        ToWin32ErrorCode := Win32ErrorCodes.ERROR_DS_DRA_OUT_OF_MEM;
    8447:
        ToWin32ErrorCode := Win32ErrorCodes.ERROR_DS_DRA_MAIL_PROBLEM;
    8448:
        ToWin32ErrorCode := Win32ErrorCodes.ERROR_DS_DRA_REF_ALREADY_EXISTS;
    8449:
        ToWin32ErrorCode := Win32ErrorCodes.ERROR_DS_DRA_REF_NOT_FOUND;
    8450:
        ToWin32ErrorCode := Win32ErrorCodes.ERROR_DS_DRA_OBJ_IS_REP_SOURCE;
    8451:
        ToWin32ErrorCode := Win32ErrorCodes.ERROR_DS_DRA_DB_ERROR;
    8452:
        ToWin32ErrorCode := Win32ErrorCodes.ERROR_DS_DRA_NO_REPLICA;
    8453:
        ToWin32ErrorCode := Win32ErrorCodes.ERROR_DS_DRA_ACCESS_DENIED;
    8454:
        ToWin32ErrorCode := Win32ErrorCodes.ERROR_DS_DRA_NOT_SUPPORTED;
    8455:
        ToWin32ErrorCode := Win32ErrorCodes.ERROR_DS_DRA_RPC_CANCELLED;
    8456:
        ToWin32ErrorCode := Win32ErrorCodes.ERROR_DS_DRA_SOURCE_DISABLED;
    8457:
        ToWin32ErrorCode := Win32ErrorCodes.ERROR_DS_DRA_SINK_DISABLED;
    8458:
        ToWin32ErrorCode := Win32ErrorCodes.ERROR_DS_DRA_NAME_COLLISION;
    8459:
        ToWin32ErrorCode := Win32ErrorCodes.ERROR_DS_DRA_SOURCE_REINSTALLED;
    8460:
        ToWin32ErrorCode := Win32ErrorCodes.ERROR_DS_DRA_MISSING_PARENT;
    8461:
        ToWin32ErrorCode := Win32ErrorCodes.ERROR_DS_DRA_PREEMPTED;
    8462:
        ToWin32ErrorCode := Win32ErrorCodes.ERROR_DS_DRA_ABANDON_SYNC;
    8463:
        ToWin32ErrorCode := Win32ErrorCodes.ERROR_DS_DRA_SHUTDOWN;
    8464:
        ToWin32ErrorCode := Win32ErrorCodes.ERROR_DS_DRA_INCOMPATIBLE_PARTIAL_SET;
    8465:
        ToWin32ErrorCode := Win32ErrorCodes.ERROR_DS_DRA_SOURCE_IS_PARTIAL_REPLICA;
    8466:
        ToWin32ErrorCode := Win32ErrorCodes.ERROR_DS_DRA_EXTN_CONNECTION_FAILED;
    8467:
        ToWin32ErrorCode := Win32ErrorCodes.ERROR_DS_INSTALL_SCHEMA_MISMATCH;
    8468:
        ToWin32ErrorCode := Win32ErrorCodes.ERROR_DS_DUP_LINK_ID;
    8469:
        ToWin32ErrorCode := Win32ErrorCodes.ERROR_DS_NAME_ERROR_RESOLVING;
    8470:
        ToWin32ErrorCode := Win32ErrorCodes.ERROR_DS_NAME_ERROR_NOT_FOUND;
    8471:
        ToWin32ErrorCode := Win32ErrorCodes.ERROR_DS_NAME_ERROR_NOT_UNIQUE;
    8472:
        ToWin32ErrorCode := Win32ErrorCodes.ERROR_DS_NAME_ERROR_NO_MAPPING;
    8473:
        ToWin32ErrorCode := Win32ErrorCodes.ERROR_DS_NAME_ERROR_DOMAIN_ONLY;
    8474:
        ToWin32ErrorCode := Win32ErrorCodes.ERROR_DS_NAME_ERROR_NO_SYNTACTICAL_MAPPING;
    8475:
        ToWin32ErrorCode := Win32ErrorCodes.ERROR_DS_CONSTRUCTED_ATT_MOD;
    8476:
        ToWin32ErrorCode := Win32ErrorCodes.ERROR_DS_WRONG_OM_OBJ_CLASS;
    8477:
        ToWin32ErrorCode := Win32ErrorCodes.ERROR_DS_DRA_REPL_PENDING;
    8478:
        ToWin32ErrorCode := Win32ErrorCodes.ERROR_DS_DS_REQUIRED;
    8479:
        ToWin32ErrorCode := Win32ErrorCodes.ERROR_DS_INVALID_LDAP_DISPLAY_NAME;
    8480:
        ToWin32ErrorCode := Win32ErrorCodes.ERROR_DS_NON_BASE_SEARCH;
    8481:
        ToWin32ErrorCode := Win32ErrorCodes.ERROR_DS_CANT_RETRIEVE_ATTS;
    8482:
        ToWin32ErrorCode := Win32ErrorCodes.ERROR_DS_BACKLINK_WITHOUT_LINK;
    8483:
        ToWin32ErrorCode := Win32ErrorCodes.ERROR_DS_EPOCH_MISMATCH;
    8484:
        ToWin32ErrorCode := Win32ErrorCodes.ERROR_DS_SRC_NAME_MISMATCH;
    8485:
        ToWin32ErrorCode := Win32ErrorCodes.ERROR_DS_SRC_AND_DST_NC_IDENTICAL;
    8486:
        ToWin32ErrorCode := Win32ErrorCodes.ERROR_DS_DST_NC_MISMATCH;
    8487:
        ToWin32ErrorCode := Win32ErrorCodes.ERROR_DS_NOT_AUTHORITIVE_FOR_DST_NC;
    8488:
        ToWin32ErrorCode := Win32ErrorCodes.ERROR_DS_SRC_GUID_MISMATCH;
    8489:
        ToWin32ErrorCode := Win32ErrorCodes.ERROR_DS_CANT_MOVE_DELETED_OBJECT;
    8490:
        ToWin32ErrorCode := Win32ErrorCodes.ERROR_DS_PDC_OPERATION_IN_PROGRESS;
    8491:
        ToWin32ErrorCode := Win32ErrorCodes.ERROR_DS_CROSS_DOMAIN_CLEANUP_REQD;
    8492:
        ToWin32ErrorCode := Win32ErrorCodes.ERROR_DS_ILLEGAL_XDOM_MOVE_OPERATION;
    8493:
        ToWin32ErrorCode := Win32ErrorCodes.ERROR_DS_CANT_WITH_ACCT_GROUP_MEMBERSHPS;
    8494:
        ToWin32ErrorCode := Win32ErrorCodes.ERROR_DS_NC_MUST_HAVE_NC_PARENT;
    8495:
        ToWin32ErrorCode := Win32ErrorCodes.ERROR_DS_CR_IMPOSSIBLE_TO_VALIDATE;
    8496:
        ToWin32ErrorCode := Win32ErrorCodes.ERROR_DS_DST_DOMAIN_NOT_NATIVE;
    8497:
        ToWin32ErrorCode := Win32ErrorCodes.ERROR_DS_MISSING_INFRASTRUCTURE_CONTAINER;
    8498:
        ToWin32ErrorCode := Win32ErrorCodes.ERROR_DS_CANT_MOVE_ACCOUNT_GROUP;
    8499:
        ToWin32ErrorCode := Win32ErrorCodes.ERROR_DS_CANT_MOVE_RESOURCE_GROUP;
    8500:
        ToWin32ErrorCode := Win32ErrorCodes.ERROR_DS_INVALID_SEARCH_FLAG;
    8501:
        ToWin32ErrorCode := Win32ErrorCodes.ERROR_DS_NO_TREE_DELETE_ABOVE_NC;
    8502:
        ToWin32ErrorCode := Win32ErrorCodes.ERROR_DS_COULDNT_LOCK_TREE_FOR_DELETE;
    8503:
        ToWin32ErrorCode := Win32ErrorCodes.ERROR_DS_COULDNT_IDENTIFY_OBJECTS_FOR_TREE_DELETE;
    8504:
        ToWin32ErrorCode := Win32ErrorCodes.ERROR_DS_SAM_INIT_FAILURE;
    8505:
        ToWin32ErrorCode := Win32ErrorCodes.ERROR_DS_SENSITIVE_GROUP_VIOLATION;
    8506:
        ToWin32ErrorCode := Win32ErrorCodes.ERROR_DS_CANT_MOD_PRIMARYGROUPID;
    8507:
        ToWin32ErrorCode := Win32ErrorCodes.ERROR_DS_ILLEGAL_BASE_SCHEMA_MOD;
    8508:
        ToWin32ErrorCode := Win32ErrorCodes.ERROR_DS_NONSAFE_SCHEMA_CHANGE;
    8509:
        ToWin32ErrorCode := Win32ErrorCodes.ERROR_DS_SCHEMA_UPDATE_DISALLOWED;
    8510:
        ToWin32ErrorCode := Win32ErrorCodes.ERROR_DS_CANT_CREATE_UNDER_SCHEMA;
    8511:
        ToWin32ErrorCode := Win32ErrorCodes.ERROR_DS_INSTALL_NO_SRC_SCH_VERSION;
    8512:
        ToWin32ErrorCode := Win32ErrorCodes.ERROR_DS_INSTALL_NO_SCH_VERSION_IN_INIFILE;
    8513:
        ToWin32ErrorCode := Win32ErrorCodes.ERROR_DS_INVALID_GROUP_TYPE;
    8514:
        ToWin32ErrorCode := Win32ErrorCodes.ERROR_DS_NO_NEST_GLOBALGROUP_IN_MIXEDDOMAIN;
    8515:
        ToWin32ErrorCode := Win32ErrorCodes.ERROR_DS_NO_NEST_LOCALGROUP_IN_MIXEDDOMAIN;
    8516:
        ToWin32ErrorCode := Win32ErrorCodes.ERROR_DS_GLOBAL_CANT_HAVE_LOCAL_MEMBER;
    8517:
        ToWin32ErrorCode := Win32ErrorCodes.ERROR_DS_GLOBAL_CANT_HAVE_UNIVERSAL_MEMBER;
    8518:
        ToWin32ErrorCode := Win32ErrorCodes.ERROR_DS_UNIVERSAL_CANT_HAVE_LOCAL_MEMBER;
    8519:
        ToWin32ErrorCode := Win32ErrorCodes.ERROR_DS_GLOBAL_CANT_HAVE_CROSSDOMAIN_MEMBER;
    8520:
        ToWin32ErrorCode := Win32ErrorCodes.ERROR_DS_LOCAL_CANT_HAVE_CROSSDOMAIN_LOCAL_MEMBER;
    8521:
        ToWin32ErrorCode := Win32ErrorCodes.ERROR_DS_HAVE_PRIMARY_MEMBERS;
    8522:
        ToWin32ErrorCode := Win32ErrorCodes.ERROR_DS_STRING_SD_CONVERSION_FAILED;
    8523:
        ToWin32ErrorCode := Win32ErrorCodes.ERROR_DS_NAMING_MASTER_GC;
    8524:
        ToWin32ErrorCode := Win32ErrorCodes.ERROR_DS_LOOKUP_FAILURE;
    8525:
        ToWin32ErrorCode := Win32ErrorCodes.ERROR_DS_COULDNT_UPDATE_SPNS;
    8526:
        ToWin32ErrorCode := Win32ErrorCodes.ERROR_DS_CANT_RETRIEVE_SD;
    8527:
        ToWin32ErrorCode := Win32ErrorCodes.ERROR_DS_KEY_NOT_UNIQUE;
    8528:
        ToWin32ErrorCode := Win32ErrorCodes.ERROR_DS_WRONG_LINKED_ATT_SYNTAX;
    8529:
        ToWin32ErrorCode := Win32ErrorCodes.ERROR_DS_SAM_NEED_BOOTKEY_PASSWORD;
    8530:
        ToWin32ErrorCode := Win32ErrorCodes.ERROR_DS_SAM_NEED_BOOTKEY_FLOPPY;
    8531:
        ToWin32ErrorCode := Win32ErrorCodes.ERROR_DS_CANT_START;
    8532:
        ToWin32ErrorCode := Win32ErrorCodes.ERROR_DS_INIT_FAILURE;
    8533:
        ToWin32ErrorCode := Win32ErrorCodes.ERROR_DS_NO_PKT_PRIVACY_ON_CONNECTION;
    8534:
        ToWin32ErrorCode := Win32ErrorCodes.ERROR_DS_SOURCE_DOMAIN_IN_FOREST;
    8535:
        ToWin32ErrorCode := Win32ErrorCodes.ERROR_DS_DESTINATION_DOMAIN_NOT_IN_FOREST;
    8536:
        ToWin32ErrorCode := Win32ErrorCodes.ERROR_DS_DESTINATION_AUDITING_NOT_ENABLED;
    8537:
        ToWin32ErrorCode := Win32ErrorCodes.ERROR_DS_CANT_FIND_DC_FOR_SRC_DOMAIN;
    8538:
        ToWin32ErrorCode := Win32ErrorCodes.ERROR_DS_SRC_OBJ_NOT_GROUP_OR_USER;
    8539:
        ToWin32ErrorCode := Win32ErrorCodes.ERROR_DS_SRC_SID_EXISTS_IN_FOREST;
    8540:
        ToWin32ErrorCode := Win32ErrorCodes.ERROR_DS_SRC_AND_DST_OBJECT_CLASS_MISMATCH;
    8541:
        ToWin32ErrorCode := Win32ErrorCodes.ERROR_SAM_INIT_FAILURE;
    8542:
        ToWin32ErrorCode := Win32ErrorCodes.ERROR_DS_DRA_SCHEMA_INFO_SHIP;
    8543:
        ToWin32ErrorCode := Win32ErrorCodes.ERROR_DS_DRA_SCHEMA_CONFLICT;
    8544:
        ToWin32ErrorCode := Win32ErrorCodes.ERROR_DS_DRA_EARLIER_SCHEMA_CONLICT;
    8545:
        ToWin32ErrorCode := Win32ErrorCodes.ERROR_DS_DRA_OBJ_NC_MISMATCH;
    8546:
        ToWin32ErrorCode := Win32ErrorCodes.ERROR_DS_NC_STILL_HAS_DSAS;
    8547:
        ToWin32ErrorCode := Win32ErrorCodes.ERROR_DS_GC_REQUIRED;
    8548:
        ToWin32ErrorCode := Win32ErrorCodes.ERROR_DS_LOCAL_MEMBER_OF_LOCAL_ONLY;
    8549:
        ToWin32ErrorCode := Win32ErrorCodes.ERROR_DS_NO_FPO_IN_UNIVERSAL_GROUPS;
    8550:
        ToWin32ErrorCode := Win32ErrorCodes.ERROR_DS_CANT_ADD_TO_GC;
    8551:
        ToWin32ErrorCode := Win32ErrorCodes.ERROR_DS_NO_CHECKPOINT_WITH_PDC;
    8552:
        ToWin32ErrorCode := Win32ErrorCodes.ERROR_DS_SOURCE_AUDITING_NOT_ENABLED;
    8553:
        ToWin32ErrorCode := Win32ErrorCodes.ERROR_DS_CANT_CREATE_IN_NONDOMAIN_NC;
    8554:
        ToWin32ErrorCode := Win32ErrorCodes.ERROR_DS_INVALID_NAME_FOR_SPN;
    8555:
        ToWin32ErrorCode := Win32ErrorCodes.ERROR_DS_FILTER_USES_CONTRUCTED_ATTRS;
    8556:
        ToWin32ErrorCode := Win32ErrorCodes.ERROR_DS_UNICODEPWD_NOT_IN_QUOTES;
    8557:
        ToWin32ErrorCode := Win32ErrorCodes.ERROR_DS_MACHINE_ACCOUNT_QUOTA_EXCEEDED;
    8558:
        ToWin32ErrorCode := Win32ErrorCodes.ERROR_DS_MUST_BE_RUN_ON_DST_DC;
    8559:
        ToWin32ErrorCode := Win32ErrorCodes.ERROR_DS_SRC_DC_MUST_BE_SP4_OR_GREATER;
    8560:
        ToWin32ErrorCode := Win32ErrorCodes.ERROR_DS_CANT_TREE_DELETE_CRITICAL_OBJ;
    8561:
        ToWin32ErrorCode := Win32ErrorCodes.ERROR_DS_INIT_FAILURE_CONSOLE;
    8562:
        ToWin32ErrorCode := Win32ErrorCodes.ERROR_DS_SAM_INIT_FAILURE_CONSOLE;
    8563:
        ToWin32ErrorCode := Win32ErrorCodes.ERROR_DS_FOREST_VERSION_TOO_HIGH;
    8564:
        ToWin32ErrorCode := Win32ErrorCodes.ERROR_DS_DOMAIN_VERSION_TOO_HIGH;
    8565:
        ToWin32ErrorCode := Win32ErrorCodes.ERROR_DS_FOREST_VERSION_TOO_LOW;
    8566:
        ToWin32ErrorCode := Win32ErrorCodes.ERROR_DS_DOMAIN_VERSION_TOO_LOW;
    8567:
        ToWin32ErrorCode := Win32ErrorCodes.ERROR_DS_INCOMPATIBLE_VERSION;
    8568:
        ToWin32ErrorCode := Win32ErrorCodes.ERROR_DS_LOW_DSA_VERSION;
    8569:
        ToWin32ErrorCode := Win32ErrorCodes.ERROR_DS_NO_BEHAVIOR_VERSION_IN_MIXEDDOMAIN;
    8570:
        ToWin32ErrorCode := Win32ErrorCodes.ERROR_DS_NOT_SUPPORTED_SORT_ORDER;
    8571:
        ToWin32ErrorCode := Win32ErrorCodes.ERROR_DS_NAME_NOT_UNIQUE;
    8572:
        ToWin32ErrorCode := Win32ErrorCodes.ERROR_DS_MACHINE_ACCOUNT_CREATED_PRENT4;
    8573:
        ToWin32ErrorCode := Win32ErrorCodes.ERROR_DS_OUT_OF_VERSION_STORE;
    8574:
        ToWin32ErrorCode := Win32ErrorCodes.ERROR_DS_INCOMPATIBLE_CONTROLS_USED;
    8575:
        ToWin32ErrorCode := Win32ErrorCodes.ERROR_DS_NO_REF_DOMAIN;
    8576:
        ToWin32ErrorCode := Win32ErrorCodes.ERROR_DS_RESERVED_LINK_ID;
    8577:
        ToWin32ErrorCode := Win32ErrorCodes.ERROR_DS_LINK_ID_NOT_AVAILABLE;
    8578:
        ToWin32ErrorCode := Win32ErrorCodes.ERROR_DS_AG_CANT_HAVE_UNIVERSAL_MEMBER;
    8579:
        ToWin32ErrorCode := Win32ErrorCodes.ERROR_DS_MODIFYDN_DISALLOWED_BY_INSTANCE_TYPE;
    8580:
        ToWin32ErrorCode := Win32ErrorCodes.ERROR_DS_NO_OBJECT_MOVE_IN_SCHEMA_NC;
    8581:
        ToWin32ErrorCode := Win32ErrorCodes.ERROR_DS_MODIFYDN_DISALLOWED_BY_FLAG;
    8582:
        ToWin32ErrorCode := Win32ErrorCodes.ERROR_DS_MODIFYDN_WRONG_GRANDPARENT;
    8583:
        ToWin32ErrorCode := Win32ErrorCodes.ERROR_DS_NAME_ERROR_TRUST_REFERRAL;
    8584:
        ToWin32ErrorCode := Win32ErrorCodes.ERROR_NOT_SUPPORTED_ON_STANDARD_SERVER;
    8585:
        ToWin32ErrorCode := Win32ErrorCodes.ERROR_DS_CANT_ACCESS_REMOTE_PART_OF_AD;
    8586:
        ToWin32ErrorCode := Win32ErrorCodes.ERROR_DS_CR_IMPOSSIBLE_TO_VALIDATE_V2;
    8587:
        ToWin32ErrorCode := Win32ErrorCodes.ERROR_DS_THREAD_LIMIT_EXCEEDED;
    8588:
        ToWin32ErrorCode := Win32ErrorCodes.ERROR_DS_NOT_CLOSEST;
    9001:
        ToWin32ErrorCode := Win32ErrorCodes.DNS_ERROR_RCODE_FORMAT_ERROR;
    9002:
        ToWin32ErrorCode := Win32ErrorCodes.DNS_ERROR_RCODE_SERVER_FAILURE;
    9003:
        ToWin32ErrorCode := Win32ErrorCodes.DNS_ERROR_RCODE_NAME_ERROR;
    9004:
        ToWin32ErrorCode := Win32ErrorCodes.DNS_ERROR_RCODE_NOT_IMPLEMENTED;
    9005:
        ToWin32ErrorCode := Win32ErrorCodes.DNS_ERROR_RCODE_REFUSED;
    9006:
        ToWin32ErrorCode := Win32ErrorCodes.DNS_ERROR_RCODE_YXDOMAIN;
    9007:
        ToWin32ErrorCode := Win32ErrorCodes.DNS_ERROR_RCODE_YXRRSET;
    9008:
        ToWin32ErrorCode := Win32ErrorCodes.DNS_ERROR_RCODE_NXRRSET;
    9009:
        ToWin32ErrorCode := Win32ErrorCodes.DNS_ERROR_RCODE_NOTAUTH;
    9010:
        ToWin32ErrorCode := Win32ErrorCodes.DNS_ERROR_RCODE_NOTZONE;
    9016:
        ToWin32ErrorCode := Win32ErrorCodes.DNS_ERROR_RCODE_BADSIG;
    9017:
        ToWin32ErrorCode := Win32ErrorCodes.DNS_ERROR_RCODE_BADKEY;
    9018:
        ToWin32ErrorCode := Win32ErrorCodes.DNS_ERROR_RCODE_BADTIME;
    9501:
        ToWin32ErrorCode := Win32ErrorCodes.DNS_INFO_NO_RECORDS;
    9502:
        ToWin32ErrorCode := Win32ErrorCodes.DNS_ERROR_BAD_PACKET;
    9503:
        ToWin32ErrorCode := Win32ErrorCodes.DNS_ERROR_NO_PACKET;
    9504:
        ToWin32ErrorCode := Win32ErrorCodes.DNS_ERROR_RCODE;
    9505:
        ToWin32ErrorCode := Win32ErrorCodes.DNS_ERROR_UNSECURE_PACKET;
    9551:
        ToWin32ErrorCode := Win32ErrorCodes.DNS_ERROR_INVALID_TYPE;
    9552:
        ToWin32ErrorCode := Win32ErrorCodes.DNS_ERROR_INVALID_IP_ADDRESS;
    9553:
        ToWin32ErrorCode := Win32ErrorCodes.DNS_ERROR_INVALID_PROPERTY;
    9554:
        ToWin32ErrorCode := Win32ErrorCodes.DNS_ERROR_TRY_AGAIN_LATER;
    9555:
        ToWin32ErrorCode := Win32ErrorCodes.DNS_ERROR_NOT_UNIQUE;
    9556:
        ToWin32ErrorCode := Win32ErrorCodes.DNS_ERROR_NON_RFC_NAME;
    9557:
        ToWin32ErrorCode := Win32ErrorCodes.DNS_STATUS_FQDN;
    9558:
        ToWin32ErrorCode := Win32ErrorCodes.DNS_STATUS_DOTTED_NAME;
    9559:
        ToWin32ErrorCode := Win32ErrorCodes.DNS_STATUS_SINGLE_PART_NAME;
    9560:
        ToWin32ErrorCode := Win32ErrorCodes.DNS_ERROR_INVALID_NAME_CHAR;
    9561:
        ToWin32ErrorCode := Win32ErrorCodes.DNS_ERROR_NUMERIC_NAME;
    9601:
        ToWin32ErrorCode := Win32ErrorCodes.DNS_ERROR_ZONE_DOES_NOT_EXIST;
    9602:
        ToWin32ErrorCode := Win32ErrorCodes.DNS_ERROR_NO_ZONE_INFO;
    9603:
        ToWin32ErrorCode := Win32ErrorCodes.DNS_ERROR_INVALID_ZONE_OPERATION;
    9604:
        ToWin32ErrorCode := Win32ErrorCodes.DNS_ERROR_ZONE_CONFIGURATION_ERROR;
    9605:
        ToWin32ErrorCode := Win32ErrorCodes.DNS_ERROR_ZONE_HAS_NO_SOA_RECORD;
    9606:
        ToWin32ErrorCode := Win32ErrorCodes.DNS_ERROR_ZONE_HAS_NO_NS_RECORDS;
    9607:
        ToWin32ErrorCode := Win32ErrorCodes.DNS_ERROR_ZONE_LOCKED;
    9608:
        ToWin32ErrorCode := Win32ErrorCodes.DNS_ERROR_ZONE_CREATION_FAILED;
    9609:
        ToWin32ErrorCode := Win32ErrorCodes.DNS_ERROR_ZONE_ALREADY_EXISTS;
    9610:
        ToWin32ErrorCode := Win32ErrorCodes.DNS_ERROR_AUTOZONE_ALREADY_EXISTS;
    9611:
        ToWin32ErrorCode := Win32ErrorCodes.DNS_ERROR_INVALID_ZONE_TYPE;
    9612:
        ToWin32ErrorCode := Win32ErrorCodes.DNS_ERROR_SECONDARY_REQUIRES_MASTER_IP;
    9613:
        ToWin32ErrorCode := Win32ErrorCodes.DNS_ERROR_ZONE_NOT_SECONDARY;
    9614:
        ToWin32ErrorCode := Win32ErrorCodes.DNS_ERROR_NEED_SECONDARY_ADDRESSES;
    9615:
        ToWin32ErrorCode := Win32ErrorCodes.DNS_ERROR_WINS_INIT_FAILED;
    9616:
        ToWin32ErrorCode := Win32ErrorCodes.DNS_ERROR_NEED_WINS_SERVERS;
    9617:
        ToWin32ErrorCode := Win32ErrorCodes.DNS_ERROR_NBSTAT_INIT_FAILED;
    9618:
        ToWin32ErrorCode := Win32ErrorCodes.DNS_ERROR_SOA_DELETE_INVALID;
    9619:
        ToWin32ErrorCode := Win32ErrorCodes.DNS_ERROR_FORWARDER_ALREADY_EXISTS;
    9651:
        ToWin32ErrorCode := Win32ErrorCodes.DNS_ERROR_PRIMARY_REQUIRES_DATAFILE;
    9652:
        ToWin32ErrorCode := Win32ErrorCodes.DNS_ERROR_INVALID_DATAFILE_NAME;
    9653:
        ToWin32ErrorCode := Win32ErrorCodes.DNS_ERROR_DATAFILE_OPEN_FAILURE;
    9654:
        ToWin32ErrorCode := Win32ErrorCodes.DNS_ERROR_FILE_WRITEBACK_FAILED;
    9655:
        ToWin32ErrorCode := Win32ErrorCodes.DNS_ERROR_DATAFILE_PARSING;
    9701:
        ToWin32ErrorCode := Win32ErrorCodes.DNS_ERROR_RECORD_DOES_NOT_EXIST;
    9702:
        ToWin32ErrorCode := Win32ErrorCodes.DNS_ERROR_RECORD_FORMAT;
    9703:
        ToWin32ErrorCode := Win32ErrorCodes.DNS_ERROR_NODE_CREATION_FAILED;
    9704:
        ToWin32ErrorCode := Win32ErrorCodes.DNS_ERROR_UNKNOWN_RECORD_TYPE;
    9705:
        ToWin32ErrorCode := Win32ErrorCodes.DNS_ERROR_RECORD_TIMED_OUT;
    9706:
        ToWin32ErrorCode := Win32ErrorCodes.DNS_ERROR_NAME_NOT_IN_ZONE;
    9707:
        ToWin32ErrorCode := Win32ErrorCodes.DNS_ERROR_CNAME_LOOP;
    9708:
        ToWin32ErrorCode := Win32ErrorCodes.DNS_ERROR_NODE_IS_CNAME;
    9709:
        ToWin32ErrorCode := Win32ErrorCodes.DNS_ERROR_CNAME_COLLISION;
    9710:
        ToWin32ErrorCode := Win32ErrorCodes.DNS_ERROR_RECORD_ONLY_AT_ZONE_ROOT;
    9711:
        ToWin32ErrorCode := Win32ErrorCodes.DNS_ERROR_RECORD_ALREADY_EXISTS;
    9712:
        ToWin32ErrorCode := Win32ErrorCodes.DNS_ERROR_SECONDARY_DATA;
    9713:
        ToWin32ErrorCode := Win32ErrorCodes.DNS_ERROR_NO_CREATE_CACHE_DATA;
    9714:
        ToWin32ErrorCode := Win32ErrorCodes.DNS_ERROR_NAME_DOES_NOT_EXIST;
    9715:
        ToWin32ErrorCode := Win32ErrorCodes.DNS_WARNING_PTR_CREATE_FAILED;
    9716:
        ToWin32ErrorCode := Win32ErrorCodes.DNS_WARNING_DOMAIN_UNDELETED;
    9717:
        ToWin32ErrorCode := Win32ErrorCodes.DNS_ERROR_DS_UNAVAILABLE;
    9718:
        ToWin32ErrorCode := Win32ErrorCodes.DNS_ERROR_DS_ZONE_ALREADY_EXISTS;
    9719:
        ToWin32ErrorCode := Win32ErrorCodes.DNS_ERROR_NO_BOOTFILE_IF_DS_ZONE;
    9751:
        ToWin32ErrorCode := Win32ErrorCodes.DNS_INFO_AXFR_COMPLETE;
    9752:
        ToWin32ErrorCode := Win32ErrorCodes.DNS_ERROR_AXFR;
    9753:
        ToWin32ErrorCode := Win32ErrorCodes.DNS_INFO_ADDED_LOCAL_WINS;
    9801:
        ToWin32ErrorCode := Win32ErrorCodes.DNS_STATUS_CONTINUE_NEEDED;
    9851:
        ToWin32ErrorCode := Win32ErrorCodes.DNS_ERROR_NO_TCPIP;
    9852:
        ToWin32ErrorCode := Win32ErrorCodes.DNS_ERROR_NO_DNS_SERVERS;
    9901:
        ToWin32ErrorCode := Win32ErrorCodes.DNS_ERROR_DP_DOES_NOT_EXIST;
    9902:
        ToWin32ErrorCode := Win32ErrorCodes.DNS_ERROR_DP_ALREADY_EXISTS;
    9903:
        ToWin32ErrorCode := Win32ErrorCodes.DNS_ERROR_DP_NOT_ENLISTED;
    9904:
        ToWin32ErrorCode := Win32ErrorCodes.DNS_ERROR_DP_ALREADY_ENLISTED;
    10004:
        ToWin32ErrorCode := Win32ErrorCodes.WSAEINTR;
    10009:
        ToWin32ErrorCode := Win32ErrorCodes.WSAEBADF;
    10013:
        ToWin32ErrorCode := Win32ErrorCodes.WSAEACCES;
    10014:
        ToWin32ErrorCode := Win32ErrorCodes.WSAEFAULT;
    10022:
        ToWin32ErrorCode := Win32ErrorCodes.WSAEINVAL;
    10024:
        ToWin32ErrorCode := Win32ErrorCodes.WSAEMFILE;
    10035:
        ToWin32ErrorCode := Win32ErrorCodes.WSAEWOULDBLOCK;
    10036:
        ToWin32ErrorCode := Win32ErrorCodes.WSAEINPROGRESS;
    10037:
        ToWin32ErrorCode := Win32ErrorCodes.WSAEALREADY;
    10038:
        ToWin32ErrorCode := Win32ErrorCodes.WSAENOTSOCK;
    10039:
        ToWin32ErrorCode := Win32ErrorCodes.WSAEDESTADDRREQ;
    10040:
        ToWin32ErrorCode := Win32ErrorCodes.WSAEMSGSIZE;
    10041:
        ToWin32ErrorCode := Win32ErrorCodes.WSAEPROTOTYPE;
    10042:
        ToWin32ErrorCode := Win32ErrorCodes.WSAENOPROTOOPT;
    10043:
        ToWin32ErrorCode := Win32ErrorCodes.WSAEPROTONOSUPPORT;
    10044:
        ToWin32ErrorCode := Win32ErrorCodes.WSAESOCKTNOSUPPORT;
    10045:
        ToWin32ErrorCode := Win32ErrorCodes.WSAEOPNOTSUPP;
    10046:
        ToWin32ErrorCode := Win32ErrorCodes.WSAEPFNOSUPPORT;
    10047:
        ToWin32ErrorCode := Win32ErrorCodes.WSAEAFNOSUPPORT;
    10048:
        ToWin32ErrorCode := Win32ErrorCodes.WSAEADDRINUSE;
    10049:
        ToWin32ErrorCode := Win32ErrorCodes.WSAEADDRNOTAVAIL;
    10050:
        ToWin32ErrorCode := Win32ErrorCodes.WSAENETDOWN;
    10051:
        ToWin32ErrorCode := Win32ErrorCodes.WSAENETUNREACH;
    10052:
        ToWin32ErrorCode := Win32ErrorCodes.WSAENETRESET;
    10053:
        ToWin32ErrorCode := Win32ErrorCodes.WSAECONNABORTED;
    10054:
        ToWin32ErrorCode := Win32ErrorCodes.WSAECONNRESET;
    10055:
        ToWin32ErrorCode := Win32ErrorCodes.WSAENOBUFS;
    10056:
        ToWin32ErrorCode := Win32ErrorCodes.WSAEISCONN;
    10057:
        ToWin32ErrorCode := Win32ErrorCodes.WSAENOTCONN;
    10058:
        ToWin32ErrorCode := Win32ErrorCodes.WSAESHUTDOWN;
    10059:
        ToWin32ErrorCode := Win32ErrorCodes.WSAETOOMANYREFS;
    10060:
        ToWin32ErrorCode := Win32ErrorCodes.WSAETIMEDOUT;
    10061:
        ToWin32ErrorCode := Win32ErrorCodes.WSAECONNREFUSED;
    10062:
        ToWin32ErrorCode := Win32ErrorCodes.WSAELOOP;
    10063:
        ToWin32ErrorCode := Win32ErrorCodes.WSAENAMETOOLONG;
    10064:
        ToWin32ErrorCode := Win32ErrorCodes.WSAEHOSTDOWN;
    10065:
        ToWin32ErrorCode := Win32ErrorCodes.WSAEHOSTUNREACH;
    10066:
        ToWin32ErrorCode := Win32ErrorCodes.WSAENOTEMPTY;
    10067:
        ToWin32ErrorCode := Win32ErrorCodes.WSAEPROCLIM;
    10068:
        ToWin32ErrorCode := Win32ErrorCodes.WSAEUSERS;
    10069:
        ToWin32ErrorCode := Win32ErrorCodes.WSAEDQUOT;
    10070:
        ToWin32ErrorCode := Win32ErrorCodes.WSAESTALE;
    10071:
        ToWin32ErrorCode := Win32ErrorCodes.WSAEREMOTE;
    10091:
        ToWin32ErrorCode := Win32ErrorCodes.WSASYSNOTREADY;
    10092:
        ToWin32ErrorCode := Win32ErrorCodes.WSAVERNOTSUPPORTED;
    10093:
        ToWin32ErrorCode := Win32ErrorCodes.WSANOTINITIALISED;
    10101:
        ToWin32ErrorCode := Win32ErrorCodes.WSAEDISCON;
    10102:
        ToWin32ErrorCode := Win32ErrorCodes.WSAENOMORE;
    10103:
        ToWin32ErrorCode := Win32ErrorCodes.WSAECANCELLED;
    10104:
        ToWin32ErrorCode := Win32ErrorCodes.WSAEINVALIDPROCTABLE;
    10105:
        ToWin32ErrorCode := Win32ErrorCodes.WSAEINVALIDPROVIDER;
    10106:
        ToWin32ErrorCode := Win32ErrorCodes.WSAEPROVIDERFAILEDINIT;
    10107:
        ToWin32ErrorCode := Win32ErrorCodes.WSASYSCALLFAILURE;
    10108:
        ToWin32ErrorCode := Win32ErrorCodes.WSASERVICE_NOT_FOUND;
    10109:
        ToWin32ErrorCode := Win32ErrorCodes.WSATYPE_NOT_FOUND;
    10110:
        ToWin32ErrorCode := Win32ErrorCodes.WSA_E_NO_MORE;
    10111:
        ToWin32ErrorCode := Win32ErrorCodes.WSA_E_CANCELLED;
    10112:
        ToWin32ErrorCode := Win32ErrorCodes.WSAEREFUSED;
    11001:
        ToWin32ErrorCode := Win32ErrorCodes.WSAHOST_NOT_FOUND;
    11002:
        ToWin32ErrorCode := Win32ErrorCodes.WSATRY_AGAIN;
    11003:
        ToWin32ErrorCode := Win32ErrorCodes.WSANO_RECOVERY;
    11004:
        ToWin32ErrorCode := Win32ErrorCodes.WSANO_DATA;
    11005:
        ToWin32ErrorCode := Win32ErrorCodes.WSA_QOS_RECEIVERS;
    11006:
        ToWin32ErrorCode := Win32ErrorCodes.WSA_QOS_SENDERS;
    11007:
        ToWin32ErrorCode := Win32ErrorCodes.WSA_QOS_NO_SENDERS;
    11008:
        ToWin32ErrorCode := Win32ErrorCodes.WSA_QOS_NO_RECEIVERS;
    11009:
        ToWin32ErrorCode := Win32ErrorCodes.WSA_QOS_REQUEST_CONFIRMED;
    11010:
        ToWin32ErrorCode := Win32ErrorCodes.WSA_QOS_ADMISSION_FAILURE;
    11011:
        ToWin32ErrorCode := Win32ErrorCodes.WSA_QOS_POLICY_FAILURE;
    11012:
        ToWin32ErrorCode := Win32ErrorCodes.WSA_QOS_BAD_STYLE;
    11013:
        ToWin32ErrorCode := Win32ErrorCodes.WSA_QOS_BAD_OBJECT;
    11014:
        ToWin32ErrorCode := Win32ErrorCodes.WSA_QOS_TRAFFIC_CTRL_ERROR;
    11015:
        ToWin32ErrorCode := Win32ErrorCodes.WSA_QOS_GENERIC_ERROR;
    11016:
        ToWin32ErrorCode := Win32ErrorCodes.WSA_QOS_ESERVICETYPE;
    11017:
        ToWin32ErrorCode := Win32ErrorCodes.WSA_QOS_EFLOWSPEC;
    11018:
        ToWin32ErrorCode := Win32ErrorCodes.WSA_QOS_EPROVSPECBUF;
    11019:
        ToWin32ErrorCode := Win32ErrorCodes.WSA_QOS_EFILTERSTYLE;
    11020:
        ToWin32ErrorCode := Win32ErrorCodes.WSA_QOS_EFILTERTYPE;
    11021:
        ToWin32ErrorCode := Win32ErrorCodes.WSA_QOS_EFILTERCOUNT;
    11022:
        ToWin32ErrorCode := Win32ErrorCodes.WSA_QOS_EOBJLENGTH;
    11023:
        ToWin32ErrorCode := Win32ErrorCodes.WSA_QOS_EFLOWCOUNT;
    11024:
        ToWin32ErrorCode := Win32ErrorCodes.WSA_QOS_EUNKNOWNPSOBJ;
    11025:
        ToWin32ErrorCode := Win32ErrorCodes.WSA_QOS_EPOLICYOBJ;
    11026:
        ToWin32ErrorCode := Win32ErrorCodes.WSA_QOS_EFLOWDESC;
    11027:
        ToWin32ErrorCode := Win32ErrorCodes.WSA_QOS_EPSFLOWSPEC;
    11028:
        ToWin32ErrorCode := Win32ErrorCodes.WSA_QOS_EPSFILTERSPEC;
    11029:
        ToWin32ErrorCode := Win32ErrorCodes.WSA_QOS_ESDMODEOBJ;
    11030:
        ToWin32ErrorCode := Win32ErrorCodes.WSA_QOS_ESHAPERATEOBJ;
    11031:
        ToWin32ErrorCode := Win32ErrorCodes.WSA_QOS_RESERVED_PETYPE;
    12000:
        ToWin32ErrorCode := Win32ErrorCodes.ERROR_SXS_SECTION_NOT_FOUND;
    12001:
        ToWin32ErrorCode := Win32ErrorCodes.ERROR_SXS_CANT_GEN_ACTCTX;
    12002:
        ToWin32ErrorCode := Win32ErrorCodes.ERROR_SXS_INVALID_ACTCTXDATA_FORMAT;
    12003:
        ToWin32ErrorCode := Win32ErrorCodes.ERROR_SXS_ASSEMBLY_NOT_FOUND;
    12004:
        ToWin32ErrorCode := Win32ErrorCodes.ERROR_SXS_MANIFEST_FORMAT_ERROR;
    12005:
        ToWin32ErrorCode := Win32ErrorCodes.ERROR_SXS_MANIFEST_PARSE_ERROR;
    12006:
        ToWin32ErrorCode := Win32ErrorCodes.ERROR_SXS_ACTIVATION_CONTEXT_DISABLED;
    12007:
        ToWin32ErrorCode := Win32ErrorCodes.ERROR_SXS_KEY_NOT_FOUND;
    12008:
        ToWin32ErrorCode := Win32ErrorCodes.ERROR_SXS_VERSION_CONFLICT;
    12009:
        ToWin32ErrorCode := Win32ErrorCodes.ERROR_SXS_WRONG_SECTION_TYPE;
    12010:
        ToWin32ErrorCode := Win32ErrorCodes.ERROR_SXS_THREAD_QUERIES_DISABLED;
    12011:
        ToWin32ErrorCode := Win32ErrorCodes.ERROR_SXS_PROCESS_DEFAULT_ALREADY_SET;
    12012:
        ToWin32ErrorCode := Win32ErrorCodes.ERROR_SXS_UNKNOWN_ENCODING_GROUP;
    12013:
        ToWin32ErrorCode := Win32ErrorCodes.ERROR_SXS_UNKNOWN_ENCODING;
    12014:
        ToWin32ErrorCode := Win32ErrorCodes.ERROR_SXS_INVALID_XML_NAMESPACE_URI;
    12015:
        ToWin32ErrorCode := Win32ErrorCodes.ERROR_SXS_ROOT_MANIFEST_DEPENDENCY_NOT_INSTALLED;
    12016:
        ToWin32ErrorCode := Win32ErrorCodes.ERROR_SXS_LEAF_MANIFEST_DEPENDENCY_NOT_INSTALLED;
    12017:
        ToWin32ErrorCode := Win32ErrorCodes.ERROR_SXS_INVALID_ASSEMBLY_IDENTITY_ATTRIBUTE;
    12018:
        ToWin32ErrorCode := Win32ErrorCodes.ERROR_SXS_MANIFEST_MISSING_REQUIRED_DEFAULT_NAMESPACE;
    12019:
        ToWin32ErrorCode := Win32ErrorCodes.ERROR_SXS_MANIFEST_INVALID_REQUIRED_DEFAULT_NAMESPACE;
    12020:
        ToWin32ErrorCode :=
            Win32ErrorCodes.ERROR_SXS_PRIVATE_MANIFEST_CROSS_PATH_WITH_REPARSE_POINT;
    12021:
        ToWin32ErrorCode := Win32ErrorCodes.ERROR_SXS_DUPLICATE_DLL_NAME;
    12022:
        ToWin32ErrorCode := Win32ErrorCodes.ERROR_SXS_DUPLICATE_WINDOWCLASS_NAME;
    12023:
        ToWin32ErrorCode := Win32ErrorCodes.ERROR_SXS_DUPLICATE_CLSID;
    12024:
        ToWin32ErrorCode := Win32ErrorCodes.ERROR_SXS_DUPLICATE_IID;
    12025:
        ToWin32ErrorCode := Win32ErrorCodes.ERROR_SXS_DUPLICATE_TLBID;
    12026:
        ToWin32ErrorCode := Win32ErrorCodes.ERROR_SXS_DUPLICATE_PROGID;
    12027:
        ToWin32ErrorCode := Win32ErrorCodes.ERROR_SXS_DUPLICATE_ASSEMBLY_NAME;
    12028:
        ToWin32ErrorCode := Win32ErrorCodes.ERROR_SXS_FILE_HASH_MISMATCH;
    12029:
        ToWin32ErrorCode := Win32ErrorCodes.ERROR_SXS_POLICY_PARSE_ERROR;
    12030:
        ToWin32ErrorCode := Win32ErrorCodes.ERROR_SXS_XML_E_MISSINGQUOTE;
    12031:
        ToWin32ErrorCode := Win32ErrorCodes.ERROR_SXS_XML_E_COMMENTSYNTAX;
    12032:
        ToWin32ErrorCode := Win32ErrorCodes.ERROR_SXS_XML_E_BADSTARTNAMECHAR;
    12033:
        ToWin32ErrorCode := Win32ErrorCodes.ERROR_SXS_XML_E_BADNAMECHAR;
    12034:
        ToWin32ErrorCode := Win32ErrorCodes.ERROR_SXS_XML_E_BADCHARINSTRING;
    12035:
        ToWin32ErrorCode := Win32ErrorCodes.ERROR_SXS_XML_E_XMLDECLSYNTAX;
    12036:
        ToWin32ErrorCode := Win32ErrorCodes.ERROR_SXS_XML_E_BADCHARDATA;
    12037:
        ToWin32ErrorCode := Win32ErrorCodes.ERROR_SXS_XML_E_MISSINGWHITESPACE;
    12038:
        ToWin32ErrorCode := Win32ErrorCodes.ERROR_SXS_XML_E_EXPECTINGTAGEND;
    12039:
        ToWin32ErrorCode := Win32ErrorCodes.ERROR_SXS_XML_E_MISSINGSEMICOLON;
    12040:
        ToWin32ErrorCode := Win32ErrorCodes.ERROR_SXS_XML_E_UNBALANCEDPAREN;
    12041:
        ToWin32ErrorCode := Win32ErrorCodes.ERROR_SXS_XML_E_INTERNALERROR;
    12042:
        ToWin32ErrorCode := Win32ErrorCodes.ERROR_SXS_XML_E_UNEXPECTED_WHITESPACE;
    12043:
        ToWin32ErrorCode := Win32ErrorCodes.ERROR_SXS_XML_E_INCOMPLETE_ENCODING;
    12044:
        ToWin32ErrorCode := Win32ErrorCodes.ERROR_SXS_XML_E_MISSING_PAREN;
    12045:
        ToWin32ErrorCode := Win32ErrorCodes.ERROR_SXS_XML_E_EXPECTINGCLOSEQUOTE;
    12046:
        ToWin32ErrorCode := Win32ErrorCodes.ERROR_SXS_XML_E_MULTIPLE_COLONS;
    12047:
        ToWin32ErrorCode := Win32ErrorCodes.ERROR_SXS_XML_E_INVALID_DECIMAL;
    12048:
        ToWin32ErrorCode := Win32ErrorCodes.ERROR_SXS_XML_E_INVALID_HEXIDECIMAL;
    12049:
        ToWin32ErrorCode := Win32ErrorCodes.ERROR_SXS_XML_E_INVALID_UNICODE;
    12050:
        ToWin32ErrorCode := Win32ErrorCodes.ERROR_SXS_XML_E_WHITESPACEORQUESTIONMARK;
    12051:
        ToWin32ErrorCode := Win32ErrorCodes.ERROR_SXS_XML_E_UNEXPECTEDENDTAG;
    12052:
        ToWin32ErrorCode := Win32ErrorCodes.ERROR_SXS_XML_E_UNCLOSEDTAG;
    12053:
        ToWin32ErrorCode := Win32ErrorCodes.ERROR_SXS_XML_E_DUPLICATEATTRIBUTE;
    12054:
        ToWin32ErrorCode := Win32ErrorCodes.ERROR_SXS_XML_E_MULTIPLEROOTS;
    12055:
        ToWin32ErrorCode := Win32ErrorCodes.ERROR_SXS_XML_E_INVALIDATROOTLEVEL;
    12056:
        ToWin32ErrorCode := Win32ErrorCodes.ERROR_SXS_XML_E_BADXMLDECL;
    12057:
        ToWin32ErrorCode := Win32ErrorCodes.ERROR_SXS_XML_E_MISSINGROOT;
    12058:
        ToWin32ErrorCode := Win32ErrorCodes.ERROR_SXS_XML_E_UNEXPECTEDEOF;
    12059:
        ToWin32ErrorCode := Win32ErrorCodes.ERROR_SXS_XML_E_BADPEREFINSUBSET;
    12060:
        ToWin32ErrorCode := Win32ErrorCodes.ERROR_SXS_XML_E_UNCLOSEDSTARTTAG;
    12061:
        ToWin32ErrorCode := Win32ErrorCodes.ERROR_SXS_XML_E_UNCLOSEDENDTAG;
    12062:
        ToWin32ErrorCode := Win32ErrorCodes.ERROR_SXS_XML_E_UNCLOSEDSTRING;
    12063:
        ToWin32ErrorCode := Win32ErrorCodes.ERROR_SXS_XML_E_UNCLOSEDCOMMENT;
    12064:
        ToWin32ErrorCode := Win32ErrorCodes.ERROR_SXS_XML_E_UNCLOSEDDECL;
    12065:
        ToWin32ErrorCode := Win32ErrorCodes.ERROR_SXS_XML_E_UNCLOSEDCDATA;
    12066:
        ToWin32ErrorCode := Win32ErrorCodes.ERROR_SXS_XML_E_RESERVEDNAMESPACE;
    12067:
        ToWin32ErrorCode := Win32ErrorCodes.ERROR_SXS_XML_E_INVALIDENCODING;
    12068:
        ToWin32ErrorCode := Win32ErrorCodes.ERROR_SXS_XML_E_INVALIDSWITCH;
    12069:
        ToWin32ErrorCode := Win32ErrorCodes.ERROR_SXS_XML_E_BADXMLCASE;
    12070:
        ToWin32ErrorCode := Win32ErrorCodes.ERROR_SXS_XML_E_INVALID_STANDALONE;
    12071:
        ToWin32ErrorCode := Win32ErrorCodes.ERROR_SXS_XML_E_UNEXPECTED_STANDALONE;
    12072:
        ToWin32ErrorCode := Win32ErrorCodes.ERROR_SXS_XML_E_INVALID_VERSION;
    12073:
        ToWin32ErrorCode := Win32ErrorCodes.ERROR_SXS_XML_E_MISSINGEQUALS;
    13000:
        ToWin32ErrorCode := Win32ErrorCodes.ERROR_IPSEC_QM_POLICY_EXISTS;
    13001:
        ToWin32ErrorCode := Win32ErrorCodes.ERROR_IPSEC_QM_POLICY_NOT_FOUND;
    13002:
        ToWin32ErrorCode := Win32ErrorCodes.ERROR_IPSEC_QM_POLICY_IN_USE;
    13003:
        ToWin32ErrorCode := Win32ErrorCodes.ERROR_IPSEC_MM_POLICY_EXISTS;
    13004:
        ToWin32ErrorCode := Win32ErrorCodes.ERROR_IPSEC_MM_POLICY_NOT_FOUND;
    13005:
        ToWin32ErrorCode := Win32ErrorCodes.ERROR_IPSEC_MM_POLICY_IN_USE;
    13006:
        ToWin32ErrorCode := Win32ErrorCodes.ERROR_IPSEC_MM_FILTER_EXISTS;
    13007:
        ToWin32ErrorCode := Win32ErrorCodes.ERROR_IPSEC_MM_FILTER_NOT_FOUND;
    13008:
        ToWin32ErrorCode := Win32ErrorCodes.ERROR_IPSEC_TRANSPORT_FILTER_EXISTS;
    13009:
        ToWin32ErrorCode := Win32ErrorCodes.ERROR_IPSEC_TRANSPORT_FILTER_NOT_FOUND;
    13010:
        ToWin32ErrorCode := Win32ErrorCodes.ERROR_IPSEC_MM_AUTH_EXISTS;
    13011:
        ToWin32ErrorCode := Win32ErrorCodes.ERROR_IPSEC_MM_AUTH_NOT_FOUND;
    13012:
        ToWin32ErrorCode := Win32ErrorCodes.ERROR_IPSEC_MM_AUTH_IN_USE;
    13013:
        ToWin32ErrorCode := Win32ErrorCodes.ERROR_IPSEC_DEFAULT_MM_POLICY_NOT_FOUND;
    13014:
        ToWin32ErrorCode := Win32ErrorCodes.ERROR_IPSEC_DEFAULT_MM_AUTH_NOT_FOUND;
    13015:
        ToWin32ErrorCode := Win32ErrorCodes.ERROR_IPSEC_DEFAULT_QM_POLICY_NOT_FOUND;
    13016:
        ToWin32ErrorCode := Win32ErrorCodes.ERROR_IPSEC_TUNNEL_FILTER_EXISTS;
    13017:
        ToWin32ErrorCode := Win32ErrorCodes.ERROR_IPSEC_TUNNEL_FILTER_NOT_FOUND;
    13018:
        ToWin32ErrorCode := Win32ErrorCodes.ERROR_IPSEC_MM_FILTER_PENDING_DELETION;
    13019:
        ToWin32ErrorCode := Win32ErrorCodes.ERROR_IPSEC_TRANSPORT_FILTER_PENDING_DELETION;
    13020:
        ToWin32ErrorCode := Win32ErrorCodes.ERROR_IPSEC_TUNNEL_FILTER_PENDING_DELETION;
    13021:
        ToWin32ErrorCode := Win32ErrorCodes.ERROR_IPSEC_MM_POLICY_PENDING_DELETION;
    13022:
        ToWin32ErrorCode := Win32ErrorCodes.ERROR_IPSEC_MM_AUTH_PENDING_DELETION;
    13023:
        ToWin32ErrorCode := Win32ErrorCodes.ERROR_IPSEC_QM_POLICY_PENDING_DELETION;
    13801:
        ToWin32ErrorCode := Win32ErrorCodes.ERROR_IPSEC_IKE_AUTH_FAIL;
    13802:
        ToWin32ErrorCode := Win32ErrorCodes.ERROR_IPSEC_IKE_ATTRIB_FAIL;
    13803:
        ToWin32ErrorCode := Win32ErrorCodes.ERROR_IPSEC_IKE_NEGOTIATION_PENDING;
    13804:
        ToWin32ErrorCode := Win32ErrorCodes.ERROR_IPSEC_IKE_GENERAL_PROCESSING_ERROR;
    13805:
        ToWin32ErrorCode := Win32ErrorCodes.ERROR_IPSEC_IKE_TIMED_OUT;
    13806:
        ToWin32ErrorCode := Win32ErrorCodes.ERROR_IPSEC_IKE_NO_CERT;
    13807:
        ToWin32ErrorCode := Win32ErrorCodes.ERROR_IPSEC_IKE_SA_DELETED;
    13808:
        ToWin32ErrorCode := Win32ErrorCodes.ERROR_IPSEC_IKE_SA_REAPED;
    13809:
        ToWin32ErrorCode := Win32ErrorCodes.ERROR_IPSEC_IKE_MM_ACQUIRE_DROP;
    13810:
        ToWin32ErrorCode := Win32ErrorCodes.ERROR_IPSEC_IKE_QM_ACQUIRE_DROP;
    13811:
        ToWin32ErrorCode := Win32ErrorCodes.ERROR_IPSEC_IKE_QUEUE_DROP_MM;
    13812:
        ToWin32ErrorCode := Win32ErrorCodes.ERROR_IPSEC_IKE_QUEUE_DROP_NO_MM;
    13813:
        ToWin32ErrorCode := Win32ErrorCodes.ERROR_IPSEC_IKE_DROP_NO_RESPONSE;
    13814:
        ToWin32ErrorCode := Win32ErrorCodes.ERROR_IPSEC_IKE_MM_DELAY_DROP;
    13815:
        ToWin32ErrorCode := Win32ErrorCodes.ERROR_IPSEC_IKE_QM_DELAY_DROP;
    13816:
        ToWin32ErrorCode := Win32ErrorCodes.ERROR_IPSEC_IKE_ERROR;
    13817:
        ToWin32ErrorCode := Win32ErrorCodes.ERROR_IPSEC_IKE_CRL_FAILED;
    13818:
        ToWin32ErrorCode := Win32ErrorCodes.ERROR_IPSEC_IKE_INVALID_KEY_USAGE;
    13819:
        ToWin32ErrorCode := Win32ErrorCodes.ERROR_IPSEC_IKE_INVALID_CERT_TYPE;
    13820:
        ToWin32ErrorCode := Win32ErrorCodes.ERROR_IPSEC_IKE_NO_PRIVATE_KEY;
    13822:
        ToWin32ErrorCode := Win32ErrorCodes.ERROR_IPSEC_IKE_DH_FAIL;
    13824:
        ToWin32ErrorCode := Win32ErrorCodes.ERROR_IPSEC_IKE_INVALID_HEADER;
    13825:
        ToWin32ErrorCode := Win32ErrorCodes.ERROR_IPSEC_IKE_NO_POLICY;
    13826:
        ToWin32ErrorCode := Win32ErrorCodes.ERROR_IPSEC_IKE_INVALID_SIGNATURE;
    13827:
        ToWin32ErrorCode := Win32ErrorCodes.ERROR_IPSEC_IKE_KERBEROS_ERROR;
    13828:
        ToWin32ErrorCode := Win32ErrorCodes.ERROR_IPSEC_IKE_NO_PUBLIC_KEY;
    13829:
        ToWin32ErrorCode := Win32ErrorCodes.ERROR_IPSEC_IKE_PROCESS_ERR;
    13830:
        ToWin32ErrorCode := Win32ErrorCodes.ERROR_IPSEC_IKE_PROCESS_ERR_SA;
    13831:
        ToWin32ErrorCode := Win32ErrorCodes.ERROR_IPSEC_IKE_PROCESS_ERR_PROP;
    13832:
        ToWin32ErrorCode := Win32ErrorCodes.ERROR_IPSEC_IKE_PROCESS_ERR_TRANS;
    13833:
        ToWin32ErrorCode := Win32ErrorCodes.ERROR_IPSEC_IKE_PROCESS_ERR_KE;
    13834:
        ToWin32ErrorCode := Win32ErrorCodes.ERROR_IPSEC_IKE_PROCESS_ERR_ID;
    13835:
        ToWin32ErrorCode := Win32ErrorCodes.ERROR_IPSEC_IKE_PROCESS_ERR_CERT;
    13836:
        ToWin32ErrorCode := Win32ErrorCodes.ERROR_IPSEC_IKE_PROCESS_ERR_CERT_REQ;
    13837:
        ToWin32ErrorCode := Win32ErrorCodes.ERROR_IPSEC_IKE_PROCESS_ERR_HASH;
    13838:
        ToWin32ErrorCode := Win32ErrorCodes.ERROR_IPSEC_IKE_PROCESS_ERR_SIG;
    13839:
        ToWin32ErrorCode := Win32ErrorCodes.ERROR_IPSEC_IKE_PROCESS_ERR_NONCE;
    13840:
        ToWin32ErrorCode := Win32ErrorCodes.ERROR_IPSEC_IKE_PROCESS_ERR_NOTIFY;
    13841:
        ToWin32ErrorCode := Win32ErrorCodes.ERROR_IPSEC_IKE_PROCESS_ERR_DELETE;
    13842:
        ToWin32ErrorCode := Win32ErrorCodes.ERROR_IPSEC_IKE_PROCESS_ERR_VENDOR;
    13843:
        ToWin32ErrorCode := Win32ErrorCodes.ERROR_IPSEC_IKE_INVALID_PAYLOAD;
    13844:
        ToWin32ErrorCode := Win32ErrorCodes.ERROR_IPSEC_IKE_LOAD_SOFT_SA;
    13845:
        ToWin32ErrorCode := Win32ErrorCodes.ERROR_IPSEC_IKE_SOFT_SA_TORN_DOWN;
    13846:
        ToWin32ErrorCode := Win32ErrorCodes.ERROR_IPSEC_IKE_INVALID_COOKIE;
    13847:
        ToWin32ErrorCode := Win32ErrorCodes.ERROR_IPSEC_IKE_NO_PEER_CERT;
    13848:
        ToWin32ErrorCode := Win32ErrorCodes.ERROR_IPSEC_IKE_PEER_CRL_FAILED;
    13849:
        ToWin32ErrorCode := Win32ErrorCodes.ERROR_IPSEC_IKE_POLICY_CHANGE;
    13850:
        ToWin32ErrorCode := Win32ErrorCodes.ERROR_IPSEC_IKE_NO_MM_POLICY;
    13851:
        ToWin32ErrorCode := Win32ErrorCodes.ERROR_IPSEC_IKE_NOTCBPRIV;
    13852:
        ToWin32ErrorCode := Win32ErrorCodes.ERROR_IPSEC_IKE_SECLOADFAIL;
    13853:
        ToWin32ErrorCode := Win32ErrorCodes.ERROR_IPSEC_IKE_FAILSSPINIT;
    13854:
        ToWin32ErrorCode := Win32ErrorCodes.ERROR_IPSEC_IKE_FAILQUERYSSP;
    13855:
        ToWin32ErrorCode := Win32ErrorCodes.ERROR_IPSEC_IKE_SRVACQFAIL;
    13856:
        ToWin32ErrorCode := Win32ErrorCodes.ERROR_IPSEC_IKE_SRVQUERYCRED;
    13857:
        ToWin32ErrorCode := Win32ErrorCodes.ERROR_IPSEC_IKE_GETSPIFAIL;
    13858:
        ToWin32ErrorCode := Win32ErrorCodes.ERROR_IPSEC_IKE_INVALID_FILTER;
    13859:
        ToWin32ErrorCode := Win32ErrorCodes.ERROR_IPSEC_IKE_OUT_OF_MEMORY;
    13860:
        ToWin32ErrorCode := Win32ErrorCodes.ERROR_IPSEC_IKE_ADD_UPDATE_KEY_FAILED;
    13861:
        ToWin32ErrorCode := Win32ErrorCodes.ERROR_IPSEC_IKE_INVALID_POLICY;
    13862:
        ToWin32ErrorCode := Win32ErrorCodes.ERROR_IPSEC_IKE_UNKNOWN_DOI;
    13863:
        ToWin32ErrorCode := Win32ErrorCodes.ERROR_IPSEC_IKE_INVALID_SITUATION;
    13864:
        ToWin32ErrorCode := Win32ErrorCodes.ERROR_IPSEC_IKE_DH_FAILURE;
    13865:
        ToWin32ErrorCode := Win32ErrorCodes.ERROR_IPSEC_IKE_INVALID_GROUP;
    13866:
        ToWin32ErrorCode := Win32ErrorCodes.ERROR_IPSEC_IKE_ENCRYPT;
    13867:
        ToWin32ErrorCode := Win32ErrorCodes.ERROR_IPSEC_IKE_DECRYPT;
    13868:
        ToWin32ErrorCode := Win32ErrorCodes.ERROR_IPSEC_IKE_POLICY_MATCH;
    13869:
        ToWin32ErrorCode := Win32ErrorCodes.ERROR_IPSEC_IKE_UNSUPPORTED_ID;
    13870:
        ToWin32ErrorCode := Win32ErrorCodes.ERROR_IPSEC_IKE_INVALID_HASH;
    13871:
        ToWin32ErrorCode := Win32ErrorCodes.ERROR_IPSEC_IKE_INVALID_HASH_ALG;
    13872:
        ToWin32ErrorCode := Win32ErrorCodes.ERROR_IPSEC_IKE_INVALID_HASH_SIZE;
    13873:
        ToWin32ErrorCode := Win32ErrorCodes.ERROR_IPSEC_IKE_INVALID_ENCRYPT_ALG;
    13874:
        ToWin32ErrorCode := Win32ErrorCodes.ERROR_IPSEC_IKE_INVALID_AUTH_ALG;
    13875:
        ToWin32ErrorCode := Win32ErrorCodes.ERROR_IPSEC_IKE_INVALID_SIG;
    13876:
        ToWin32ErrorCode := Win32ErrorCodes.ERROR_IPSEC_IKE_LOAD_FAILED;
    13877:
        ToWin32ErrorCode := Win32ErrorCodes.ERROR_IPSEC_IKE_RPC_DELETE;
    13878:
        ToWin32ErrorCode := Win32ErrorCodes.ERROR_IPSEC_IKE_BENIGN_REINIT;
    13879:
        ToWin32ErrorCode := Win32ErrorCodes.ERROR_IPSEC_IKE_INVALID_RESPONDER_LIFETIME_NOTIFY;
    13880:
        ToWin32ErrorCode := Win32ErrorCodes.ERROR_IPSEC_IKE_QM_LIMIT_REAP;
    13881:
        ToWin32ErrorCode := Win32ErrorCodes.ERROR_IPSEC_IKE_INVALID_CERT_KEYLEN;
    13882:
        ToWin32ErrorCode := Win32ErrorCodes.ERROR_IPSEC_IKE_MM_LIMIT;
    13883:
        ToWin32ErrorCode := Win32ErrorCodes.ERROR_IPSEC_IKE_NEGOTIATION_DISABLED;
    13884:
        ToWin32ErrorCode := Win32ErrorCodes.ERROR_IPSEC_IKE_QM_LIMIT;
ELSE
    ToWin32ErrorCode := Win32ErrorCodes.ERR_UNKNOWN;
END_CASE

END_FUNCTION

// ---- Win32_Tests/Win32ErrorCodeDesciption_Tests.TcPOU
{attribute 'hide'}
FUNCTION_BLOCK Win32ErrorCodeDesciption_Tests EXTENDS TcUnit.FB_TestSuite

DescriptionOfKnownErrorCode();
DescriptionOfUnknownErrorCode();

METHOD DescriptionOfKnownErrorCode
TcUnit.TEST('DescriptionOfKnownErrorCode');

AssertEquals_STRING(
    Expected:='The system cannot find the file specified.',
    Actual:=Win32ErrorCodeDescription(Win32ErrorCodes.ERROR_FILE_NOT_FOUND),
    Message:='Error description not correct.'
);

TcUnit.TEST_FINISHED();
END_METHOD

METHOD DescriptionOfUnknownErrorCode
TcUnit.TEST('DescriptionOfUnknownErrorCode');

AssertEquals_STRING(
    Expected:='Unknown Win32 error code.',
    Actual:=Win32ErrorCodeDescription(Win32ErrorCodes.ERR_UNKNOWN),
    Message:='Error description not correct.'
);

TcUnit.TEST_FINISHED();
END_METHOD

END_FUNCTION_BLOCK

// ---- Win32/Win32ErrorCodeDescription.TcPOU
(*
Returns an description of the error from the Win32ErrorCodes datatype.

## Example
```
win32ErrorCode := Win32ErrorCodes.ERROR_CANNOT_MAKE;
errorDescription := Win32ErrorCodeDescription(win32ErrorCode); // 'The directory or file cannot be created.'
```

## Source
https://infosys.beckhoff.com/content/1033/devicemanager/391166347.html?id=8711134805786442486
*)
FUNCTION Win32ErrorCodeDescription : T_MaxString
VAR_INPUT
    win32ErrorCode : Win32ErrorCodes;
END_VAR

CASE win32ErrorCode OF
    Win32ErrorCodes.ERROR_SUCCESS:
        Win32ErrorCodeDescription := 'The operation completed successfully.';
    Win32ErrorCodes.ERROR_INVALID_FUNCTION:
        Win32ErrorCodeDescription := 'Incorrect function.';
    Win32ErrorCodes.ERROR_FILE_NOT_FOUND:
        Win32ErrorCodeDescription := 'The system cannot find the file specified.';
    Win32ErrorCodes.ERROR_PATH_NOT_FOUND:
        Win32ErrorCodeDescription := 'The system cannot find the path specified.';
    Win32ErrorCodes.ERROR_TOO_MANY_OPEN_FILES:
        Win32ErrorCodeDescription := 'The system cannot open the file.';
    Win32ErrorCodes.ERROR_ACCESS_DENIED:
        Win32ErrorCodeDescription := 'Access is denied.';
    Win32ErrorCodes.ERROR_INVALID_HANDLE:
        Win32ErrorCodeDescription := 'The handle is invalid.';
    Win32ErrorCodes.ERROR_ARENA_TRASHED:
        Win32ErrorCodeDescription := 'The storage control blocks were destroyed.';
    Win32ErrorCodes.ERROR_NOT_ENOUGH_MEMORY:
        Win32ErrorCodeDescription := 'Not enough storage is available to process this command.';
    Win32ErrorCodes.ERROR_INVALID_BLOCK:
        Win32ErrorCodeDescription := 'The storage control block address is invalid.';
    Win32ErrorCodes.ERROR_BAD_ENVIRONMENT:
        Win32ErrorCodeDescription := 'The environment is incorrect.';
    Win32ErrorCodes.ERROR_BAD_FORMAT:
        Win32ErrorCodeDescription :=
            'An attempt was made to load a program with an incorrect format.';
    Win32ErrorCodes.ERROR_INVALID_ACCESS:
        Win32ErrorCodeDescription := 'The access code is invalid.';
    Win32ErrorCodes.ERROR_INVALID_DATA:
        Win32ErrorCodeDescription := 'The data is invalid.';
    Win32ErrorCodes.ERROR_OUTOFMEMORY:
        Win32ErrorCodeDescription := 'Not enough storage is available to complete this operation.';
    Win32ErrorCodes.ERROR_INVALID_DRIVE:
        Win32ErrorCodeDescription := 'The system cannot find the drive specified.';
    Win32ErrorCodes.ERROR_CURRENT_DIRECTORY:
        Win32ErrorCodeDescription := 'The directory cannot be removed.';
    Win32ErrorCodes.ERROR_NOT_SAME_DEVICE:
        Win32ErrorCodeDescription := 'The system cannot move the file to a different disk drive.';
    Win32ErrorCodes.ERROR_NO_MORE_FILES:
        Win32ErrorCodeDescription := 'There are no more files.';
    Win32ErrorCodes.ERROR_WRITE_PROTECT:
        Win32ErrorCodeDescription := 'The media is write protected.';
    Win32ErrorCodes.ERROR_BAD_UNIT:
        Win32ErrorCodeDescription := 'The system cannot find the device specified.';
    Win32ErrorCodes.ERROR_NOT_READY:
        Win32ErrorCodeDescription := 'The device is not ready.';
    Win32ErrorCodes.ERROR_BAD_COMMAND:
        Win32ErrorCodeDescription := 'The device does not recognize the command.';
    Win32ErrorCodes.ERROR_CRC:
        Win32ErrorCodeDescription := 'Data error (cyclic redundancy check).';
    Win32ErrorCodes.ERROR_BAD_LENGTH:
        Win32ErrorCodeDescription :=
            'The program issued a command but the command length is incorrect.';
    Win32ErrorCodes.ERROR_SEEK:
        Win32ErrorCodeDescription :=
            'The drive cannot locate a specific area or track on the disk.';
    Win32ErrorCodes.ERROR_NOT_DOS_DISK:
        Win32ErrorCodeDescription := 'The specified disk or diskette cannot be accessed.';
    Win32ErrorCodes.ERROR_SECTOR_NOT_FOUND:
        Win32ErrorCodeDescription := 'The drive cannot find the sector requested.';
    Win32ErrorCodes.ERROR_OUT_OF_PAPER:
        Win32ErrorCodeDescription := 'The printer is out of paper.';
    Win32ErrorCodes.ERROR_WRITE_FAULT:
        Win32ErrorCodeDescription := 'The system cannot write to the specified device.';
    Win32ErrorCodes.ERROR_READ_FAULT:
        Win32ErrorCodeDescription := 'The system cannot read from the specified device.';
    Win32ErrorCodes.ERROR_GEN_FAILURE:
        Win32ErrorCodeDescription := 'A device attached to the system is not functioning.';
    Win32ErrorCodes.ERROR_SHARING_VIOLATION:
        Win32ErrorCodeDescription :=
            'The process cannot access the file because it is being used by another process.';
    Win32ErrorCodes.ERROR_LOCK_VIOLATION:
        Win32ErrorCodeDescription := 'The process cannot access the file because another process has locked a portion of the file.';
    Win32ErrorCodes.ERROR_WRONG_DISK:
        Win32ErrorCodeDescription :=
            'The wrong diskette is in the drive. Insert %2 (Volume Serial Number: %3) into drive %1.';
    Win32ErrorCodes.ERROR_SHARING_BUFFER_EXCEEDED:
        Win32ErrorCodeDescription := 'Too many files opened for sharing.';
    Win32ErrorCodes.ERROR_HANDLE_EOF:
        Win32ErrorCodeDescription := 'Reached the end of the file.';
    Win32ErrorCodes.ERROR_HANDLE_DISK_FULL:
        Win32ErrorCodeDescription := 'The disk is full.';
    Win32ErrorCodes.ERROR_NOT_SUPPORTED:
        Win32ErrorCodeDescription := 'The request is not supported.';
    Win32ErrorCodes.ERROR_REM_NOT_LIST:
        Win32ErrorCodeDescription := 'The remote computer is not available.';
    Win32ErrorCodes.ERROR_DUP_NAME:
        Win32ErrorCodeDescription := 'A duplicate name exists on the network.';
    Win32ErrorCodes.ERROR_BAD_NETPATH:
        Win32ErrorCodeDescription := 'The network path was not found.';
    Win32ErrorCodes.ERROR_NETWORK_BUSY:
        Win32ErrorCodeDescription := 'The network is busy.';
    Win32ErrorCodes.ERROR_DEV_NOT_EXIST:
        Win32ErrorCodeDescription :=
            'The specified network resource or device is no longer available.';
    Win32ErrorCodes.ERROR_TOO_MANY_CMDS:
        Win32ErrorCodeDescription := 'The network BIOS command limit has been reached.';
    Win32ErrorCodes.ERROR_ADAP_HDW_ERR:
        Win32ErrorCodeDescription := 'A network adapter hardware error occurred.';
    Win32ErrorCodes.ERROR_BAD_NET_RESP:
        Win32ErrorCodeDescription :=
            'The specified server cannot perform the requested operation.';
    Win32ErrorCodes.ERROR_UNEXP_NET_ERR:
        Win32ErrorCodeDescription := 'An unexpected network error occurred.';
    Win32ErrorCodes.ERROR_BAD_REM_ADAP:
        Win32ErrorCodeDescription := 'The remote adapter is not compatible.';
    Win32ErrorCodes.ERROR_PRINTQ_FULL:
        Win32ErrorCodeDescription := 'The printer queue is full.';
    Win32ErrorCodes.ERROR_NO_SPOOL_SPACE:
        Win32ErrorCodeDescription :=
            'Space to store the file waiting to be printed is not available on the server.';
    Win32ErrorCodes.ERROR_PRINT_CANCELLED:
        Win32ErrorCodeDescription := 'Your file waiting to be printed was deleted.';
    Win32ErrorCodes.ERROR_NETNAME_DELETED:
        Win32ErrorCodeDescription := 'The specified network name is no longer available.';
    Win32ErrorCodes.ERROR_NETWORK_ACCESS_DENIED:
        Win32ErrorCodeDescription := 'Network access is denied.';
    Win32ErrorCodes.ERROR_BAD_DEV_TYPE:
        Win32ErrorCodeDescription := 'The network resource type is not correct.';
    Win32ErrorCodes.ERROR_BAD_NET_NAME:
        Win32ErrorCodeDescription := 'The network name cannot be found.';
    Win32ErrorCodes.ERROR_TOO_MANY_NAMES:
        Win32ErrorCodeDescription :=
            'The name limit for the local computer network adapter card was exceeded.';
    Win32ErrorCodes.ERROR_TOO_MANY_SESS:
        Win32ErrorCodeDescription := 'The network BIOS session limit was exceeded.';
    Win32ErrorCodes.ERROR_SHARING_PAUSED:
        Win32ErrorCodeDescription :=
            'The remote server has been paused or is in the process of being started.';
    Win32ErrorCodes.ERROR_REQ_NOT_ACCEP:
        Win32ErrorCodeDescription := 'No more connections can be made to this remote computer at this time because there are already as many connections as the computer can accept.';
    Win32ErrorCodes.ERROR_REDIR_PAUSED:
        Win32ErrorCodeDescription := 'The specified printer or disk device has been paused.';
    Win32ErrorCodes.ERROR_FILE_EXISTS:
        Win32ErrorCodeDescription := 'The file exists.';
    Win32ErrorCodes.ERROR_CANNOT_MAKE:
        Win32ErrorCodeDescription := 'The directory or file cannot be created.';
    Win32ErrorCodes.ERROR_FAIL_I24:
        Win32ErrorCodeDescription := 'Fail on INT 24.';
    Win32ErrorCodes.ERROR_OUT_OF_STRUCTURES:
        Win32ErrorCodeDescription := 'Storage to process this request is not available.';
    Win32ErrorCodes.ERROR_ALREADY_ASSIGNED:
        Win32ErrorCodeDescription := 'The local device name is already in use.';
    Win32ErrorCodes.ERROR_INVALID_PASSWORD:
        Win32ErrorCodeDescription := 'The specified network password is not correct.';
    Win32ErrorCodes.ERROR_INVALID_PARAMETER:
        Win32ErrorCodeDescription := 'The parameter is incorrect.';
    Win32ErrorCodes.ERROR_NET_WRITE_FAULT:
        Win32ErrorCodeDescription := 'A write fault occurred on the network.';
    Win32ErrorCodes.ERROR_NO_PROC_SLOTS:
        Win32ErrorCodeDescription := 'The system cannot start another process at this time.';
    Win32ErrorCodes.ERROR_TOO_MANY_SEMAPHORES:
        Win32ErrorCodeDescription := 'Cannot create another system semaphore.';
    Win32ErrorCodes.ERROR_EXCL_SEM_ALREADY_OWNED:
        Win32ErrorCodeDescription := 'The exclusive semaphore is owned by another process.';
    Win32ErrorCodes.ERROR_SEM_IS_SET:
        Win32ErrorCodeDescription := 'The semaphore is set and cannot be closed.';
    Win32ErrorCodes.ERROR_TOO_MANY_SEM_REQUESTS:
        Win32ErrorCodeDescription := 'The semaphore cannot be set again.';
    Win32ErrorCodes.ERROR_INVALID_AT_INTERRUPT_TIME:
        Win32ErrorCodeDescription := 'Cannot request exclusive semaphores at interrupt time.';
    Win32ErrorCodes.ERROR_SEM_OWNER_DIED:
        Win32ErrorCodeDescription := 'The previous ownership of this semaphore has ended.';
    Win32ErrorCodes.ERROR_SEM_USER_LIMIT:
        Win32ErrorCodeDescription := 'Insert the diskette for drive %1.';
    Win32ErrorCodes.ERROR_DISK_CHANGE:
        Win32ErrorCodeDescription :=
            'The program stopped because an alternate diskette was not inserted.';
    Win32ErrorCodes.ERROR_DRIVE_LOCKED:
        Win32ErrorCodeDescription := 'The disk is in use or locked by another process.';
    Win32ErrorCodes.ERROR_BROKEN_PIPE:
        Win32ErrorCodeDescription := 'The pipe has been ended.';
    Win32ErrorCodes.ERROR_OPEN_FAILED:
        Win32ErrorCodeDescription := 'The system cannot open the device or file specified.';
    Win32ErrorCodes.ERROR_BUFFER_OVERFLOW:
        Win32ErrorCodeDescription := 'The file name is too long.';
    Win32ErrorCodes.ERROR_DISK_FULL:
        Win32ErrorCodeDescription := 'There is not enough space on the disk.';
    Win32ErrorCodes.ERROR_NO_MORE_SEARCH_HANDLES:
        Win32ErrorCodeDescription := 'No more internal file identifiers available.';
    Win32ErrorCodes.ERROR_INVALID_TARGET_HANDLE:
        Win32ErrorCodeDescription := 'The target internal file identifier is incorrect.';
    Win32ErrorCodes.ERROR_INVALID_CATEGORY:
        Win32ErrorCodeDescription :=
            'The IOCTL call made by the application program is not correct.';
    Win32ErrorCodes.ERROR_INVALID_VERIFY_SWITCH:
        Win32ErrorCodeDescription := 'The verify-on-write switch parameter value is not correct.';
    Win32ErrorCodes.ERROR_BAD_DRIVER_LEVEL:
        Win32ErrorCodeDescription := 'The system does not support the command requested.';
    Win32ErrorCodes.ERROR_CALL_NOT_IMPLEMENTED:
        Win32ErrorCodeDescription := 'This function is not supported on this system.';
    Win32ErrorCodes.ERROR_SEM_TIMEOUT:
        Win32ErrorCodeDescription := 'The semaphore timeout period has expired.';
    Win32ErrorCodes.ERROR_INSUFFICIENT_BUFFER:
        Win32ErrorCodeDescription := 'The data area passed to a system call is too small.';
    Win32ErrorCodes.ERROR_INVALID_NAME:
        Win32ErrorCodeDescription :=
            'The filename, directory name, or volume label syntax is incorrect.';
    Win32ErrorCodes.ERROR_INVALID_LEVEL:
        Win32ErrorCodeDescription := 'The system call level is not correct.';
    Win32ErrorCodes.ERROR_NO_VOLUME_LABEL:
        Win32ErrorCodeDescription := 'The disk has no volume label.';
    Win32ErrorCodes.ERROR_MOD_NOT_FOUND:
        Win32ErrorCodeDescription := 'The specified module could not be found.';
    Win32ErrorCodes.ERROR_PROC_NOT_FOUND:
        Win32ErrorCodeDescription := 'The specified procedure could not be found.';
    Win32ErrorCodes.ERROR_WAIT_NO_CHILDREN:
        Win32ErrorCodeDescription := 'There are no child processes to wait for.';
    Win32ErrorCodes.ERROR_CHILD_NOT_COMPLETE:
        Win32ErrorCodeDescription := 'The %1 application cannot be run in Win32 mode.';
    Win32ErrorCodes.ERROR_DIRECT_ACCESS_HANDLE:
        Win32ErrorCodeDescription := 'Attempt to use a file handle to an open disk partition for an operation other than raw disk I/O.';
    Win32ErrorCodes.ERROR_NEGATIVE_SEEK:
        Win32ErrorCodeDescription :=
            'An attempt was made to move the file pointer before the beginning of the file.';
    Win32ErrorCodes.ERROR_SEEK_ON_DEVICE:
        Win32ErrorCodeDescription :=
            'The file pointer cannot be set on the specified device or file.';
    Win32ErrorCodes.ERROR_IS_JOIN_TARGET:
        Win32ErrorCodeDescription := 'A JOIN or SUBST command cannot be used for a drive that contains previously joined drives.';
    Win32ErrorCodes.ERROR_IS_JOINED:
        Win32ErrorCodeDescription := 'An attempt was made to use a JOIN or SUBST command on a drive that has already been joined.';
    Win32ErrorCodes.ERROR_IS_SUBSTED:
        Win32ErrorCodeDescription := 'An attempt was made to use a JOIN or SUBST command on a drive that has already been substituted.';
    Win32ErrorCodes.ERROR_NOT_JOINED:
        Win32ErrorCodeDescription :=
            'The system tried to delete the JOIN of a drive that is not joined.';
    Win32ErrorCodes.ERROR_NOT_SUBSTED:
        Win32ErrorCodeDescription :=
            'The system tried to delete the substitution of a drive that is not substituted.';
    Win32ErrorCodes.ERROR_JOIN_TO_JOIN:
        Win32ErrorCodeDescription :=
            'The system tried to join a drive to a directory on a joined drive.';
    Win32ErrorCodes.ERROR_SUBST_TO_SUBST:
        Win32ErrorCodeDescription :=
            'The system tried to substitute a drive to a directory on a substituted drive.';
    Win32ErrorCodes.ERROR_JOIN_TO_SUBST:
        Win32ErrorCodeDescription :=
            'The system tried to join a drive to a directory on a substituted drive.';
    Win32ErrorCodes.ERROR_SUBST_TO_JOIN:
        Win32ErrorCodeDescription :=
            'The system tried to SUBST a drive to a directory on a joined drive.';
    Win32ErrorCodes.ERROR_BUSY_DRIVE:
        Win32ErrorCodeDescription := 'The system cannot perform a JOIN or SUBST at this time.';
    Win32ErrorCodes.ERROR_SAME_DRIVE:
        Win32ErrorCodeDescription :=
            'The system cannot join or substitute a drive to or for a directory on the same drive.';
    Win32ErrorCodes.ERROR_DIR_NOT_ROOT:
        Win32ErrorCodeDescription := 'The directory is not a subdirectory of the root directory.';
    Win32ErrorCodes.ERROR_DIR_NOT_EMPTY:
        Win32ErrorCodeDescription := 'The directory is not empty.';
    Win32ErrorCodes.ERROR_IS_SUBST_PATH:
        Win32ErrorCodeDescription := 'The path specified is being used in a substitute.';
    Win32ErrorCodes.ERROR_IS_JOIN_PATH:
        Win32ErrorCodeDescription := 'Not enough resources are available to process this command.';
    Win32ErrorCodes.ERROR_PATH_BUSY:
        Win32ErrorCodeDescription := 'The path specified cannot be used at this time.';
    Win32ErrorCodes.ERROR_IS_SUBST_TARGET:
        Win32ErrorCodeDescription := 'An attempt was made to join or substitute a drive for which a directory on the drive is the target of a previous substitute.';
    Win32ErrorCodes.ERROR_SYSTEM_TRACE:
        Win32ErrorCodeDescription := 'System trace information was not specified in your CONFIG.SYS file, or tracing is disallowed.';
    Win32ErrorCodes.ERROR_INVALID_EVENT_COUNT:
        Win32ErrorCodeDescription :=
            'The number of specified semaphore events for DosMuxSemWait is not correct.';
    Win32ErrorCodes.ERROR_TOO_MANY_MUXWAITERS:
        Win32ErrorCodeDescription :=
            'DosMuxSemWait did not execute; too many semaphores are already set.';
    Win32ErrorCodes.ERROR_INVALID_LIST_FORMAT:
        Win32ErrorCodeDescription := 'The DosMuxSemWait list is not correct.';
    Win32ErrorCodes.ERROR_LABEL_TOO_LONG:
        Win32ErrorCodeDescription :=
            'The volume label you entered exceeds the label character limit of the target file system.';
    Win32ErrorCodes.ERROR_TOO_MANY_TCBS:
        Win32ErrorCodeDescription := 'Cannot create another thread.';
    Win32ErrorCodes.ERROR_SIGNAL_REFUSED:
        Win32ErrorCodeDescription := 'The recipient process has refused the signal.';
    Win32ErrorCodes.ERROR_DISCARDED:
        Win32ErrorCodeDescription := 'The segment is already discarded and cannot be locked.';
    Win32ErrorCodes.ERROR_NOT_LOCKED:
        Win32ErrorCodeDescription := 'The segment is already unlocked.';
    Win32ErrorCodes.ERROR_BAD_THREADID_ADDR:
        Win32ErrorCodeDescription := 'The address for the thread ID is not correct.';
    Win32ErrorCodes.ERROR_BAD_ARGUMENTS:
        Win32ErrorCodeDescription := 'The argument string passed to DosExecPgm is not correct.';
    Win32ErrorCodes.ERROR_BAD_PATHNAME:
        Win32ErrorCodeDescription := 'The specified path is invalid.';
    Win32ErrorCodes.ERROR_SIGNAL_PENDING:
        Win32ErrorCodeDescription := 'A signal is already pending.';
    Win32ErrorCodes.ERROR_MAX_THRDS_REACHED:
        Win32ErrorCodeDescription := 'No more threads can be created in the system.';
    Win32ErrorCodes.ERROR_LOCK_FAILED:
        Win32ErrorCodeDescription := 'Unable to lock a region of a file.';
    Win32ErrorCodes.ERROR_BUSY:
        Win32ErrorCodeDescription := 'The requested resource is in use.';
    Win32ErrorCodes.ERROR_CANCEL_VIOLATION:
        Win32ErrorCodeDescription :=
            'A lock request was not outstanding for the supplied cancel region.';
    Win32ErrorCodes.ERROR_ATOMIC_LOCKS_NOT_SUPPORTED:
        Win32ErrorCodeDescription :=
            'The file system does not support atomic changes to the lock type.';
    Win32ErrorCodes.ERROR_INVALID_SEGMENT_NUMBER:
        Win32ErrorCodeDescription := 'The system detected a segment number that was not correct.';
    Win32ErrorCodes.ERROR_INVALID_ORDINAL:
        Win32ErrorCodeDescription := 'The operating system cannot run %1.';
    Win32ErrorCodes.ERROR_ALREADY_EXISTS:
        Win32ErrorCodeDescription := 'Cannot create a file when that file already exists.';
    Win32ErrorCodes.ERROR_INVALID_FLAG_NUMBER:
        Win32ErrorCodeDescription := 'The flag passed is not correct.';
    Win32ErrorCodes.ERROR_SEM_NOT_FOUND:
        Win32ErrorCodeDescription := 'The specified system semaphore name was not found.';
    Win32ErrorCodes.ERROR_INVALID_STARTING_CODESEG:
        Win32ErrorCodeDescription := 'The operating system cannot run %1.';
    Win32ErrorCodes.ERROR_INVALID_STACKSEG:
        Win32ErrorCodeDescription := 'The operating system cannot run %1.';
    Win32ErrorCodes.ERROR_INVALID_MODULETYPE:
        Win32ErrorCodeDescription := 'The operating system cannot run %1.';
    Win32ErrorCodes.ERROR_INVALID_EXE_SIGNATURE:
        Win32ErrorCodeDescription := 'Cannot run %1 in Win32 mode.';
    Win32ErrorCodes.ERROR_EXE_MARKED_INVALID:
        Win32ErrorCodeDescription := 'The operating system cannot run %1.';
    Win32ErrorCodes.ERROR_BAD_EXE_FORMAT:
        Win32ErrorCodeDescription := '%1 is not a valid Win32 application.';
    Win32ErrorCodes.ERROR_ITERATED_DATA_EXCEEDS_64k:
        Win32ErrorCodeDescription := 'The operating system cannot run %1.';
    Win32ErrorCodes.ERROR_INVALID_MINALLOCSIZE:
        Win32ErrorCodeDescription := 'The operating system cannot run %1.';
    Win32ErrorCodes.ERROR_DYNLINK_FROM_INVALID_RING:
        Win32ErrorCodeDescription := 'The operating system cannot run this application program.';
    Win32ErrorCodes.ERROR_IOPL_NOT_ENABLED:
        Win32ErrorCodeDescription :=
            'The operating system is not presently configured to run this application.';
    Win32ErrorCodes.ERROR_INVALID_SEGDPL:
        Win32ErrorCodeDescription := 'The operating system cannot run %1.';
    Win32ErrorCodes.ERROR_AUTODATASEG_EXCEEDS_64k:
        Win32ErrorCodeDescription := 'The operating system cannot run this application program.';
    Win32ErrorCodes.ERROR_RING2SEG_MUST_BE_MOVABLE:
        Win32ErrorCodeDescription := 'The code segment cannot be greater than or equal to 64K.';
    Win32ErrorCodes.ERROR_RELOC_CHAIN_XEEDS_SEGLIM:
        Win32ErrorCodeDescription := 'The operating system cannot run %1.';
    Win32ErrorCodes.ERROR_INFLOOP_IN_RELOC_CHAIN:
        Win32ErrorCodeDescription := 'The operating system cannot run %1.';
    Win32ErrorCodes.ERROR_ENVVAR_NOT_FOUND:
        Win32ErrorCodeDescription :=
            'The system could not find the environment option that was entered.';
    Win32ErrorCodes.ERROR_NO_SIGNAL_SENT:
        Win32ErrorCodeDescription := 'No process in the command subtree has a signal handler.';
    Win32ErrorCodes.ERROR_FILENAME_EXCED_RANGE:
        Win32ErrorCodeDescription := 'The filename or extension is too long.';
    Win32ErrorCodes.ERROR_RING2_STACK_IN_USE:
        Win32ErrorCodeDescription := 'The ring 2 stack is in use.';
    Win32ErrorCodes.ERROR_META_EXPANSION_TOO_LONG:
        Win32ErrorCodeDescription := 'The global filename characters, * or ?, are entered incorrectly or too many global filename characters are specified.';
    Win32ErrorCodes.ERROR_INVALID_SIGNAL_NUMBER:
        Win32ErrorCodeDescription := 'The signal being posted is not correct.';
    Win32ErrorCodes.ERROR_THREAD_1_INACTIVE:
        Win32ErrorCodeDescription := 'The signal handler cannot be set.';
    Win32ErrorCodes.ERROR_LOCKED:
        Win32ErrorCodeDescription := 'The segment is locked and cannot be reallocated.';
    Win32ErrorCodes.ERROR_TOO_MANY_MODULES:
        Win32ErrorCodeDescription :=
            'Too many dynamic-link modules are attached to this program or dynamic-link module.';
    Win32ErrorCodes.ERROR_NESTING_NOT_ALLOWED:
        Win32ErrorCodeDescription := 'Cannot nest calls to LoadModule.';
    Win32ErrorCodes.ERROR_EXE_MACHINE_TYPE_MISMATCH:
        Win32ErrorCodeDescription :=
            'The image file %1 is valid, but is for a machine type other than the current machine.';
    Win32ErrorCodes.ERROR_BAD_PIPE:
        Win32ErrorCodeDescription := 'The pipe state is invalid.';
    Win32ErrorCodes.ERROR_PIPE_BUSY:
        Win32ErrorCodeDescription := 'All pipe instances are busy.';
    Win32ErrorCodes.ERROR_NO_DATA:
        Win32ErrorCodeDescription := 'The pipe is being closed.';
    Win32ErrorCodes.ERROR_PIPE_NOT_CONNECTED:
        Win32ErrorCodeDescription := 'No process is on the other end of the pipe.';
    Win32ErrorCodes.ERROR_MORE_DATA:
        Win32ErrorCodeDescription := 'More data is available.';
    Win32ErrorCodes.ERROR_VC_DISCONNECTED:
        Win32ErrorCodeDescription := 'The session was canceled.';
    Win32ErrorCodes.ERROR_INVALID_EA_NAME:
        Win32ErrorCodeDescription := 'The specified extended attribute name was invalid.';
    Win32ErrorCodes.ERROR_EA_LIST_INCONSISTENT:
        Win32ErrorCodeDescription := 'The extended attributes are inconsistent.';
    Win32ErrorCodes.WAIT_TIMEOUT:
        Win32ErrorCodeDescription := 'The wait operation timed out.';
    Win32ErrorCodes.ERROR_NO_MORE_ITEMS:
        Win32ErrorCodeDescription := 'No more data is available.';
    Win32ErrorCodes.ERROR_CANNOT_COPY:
        Win32ErrorCodeDescription := 'The copy functions cannot be used.';
    Win32ErrorCodes.ERROR_DIRECTORY:
        Win32ErrorCodeDescription := 'The directory name is invalid.';
    Win32ErrorCodes.ERROR_EAS_DIDNT_FIT:
        Win32ErrorCodeDescription := 'The extended attributes did not fit in the buffer.';
    Win32ErrorCodes.ERROR_EA_FILE_CORRUPT:
        Win32ErrorCodeDescription :=
            'The extended attribute file on the mounted file system is corrupt.';
    Win32ErrorCodes.ERROR_EA_TABLE_FULL:
        Win32ErrorCodeDescription := 'The extended attribute table file is full.';
    Win32ErrorCodes.ERROR_INVALID_EA_HANDLE:
        Win32ErrorCodeDescription := 'The specified extended attribute handle is invalid.';
    Win32ErrorCodes.ERROR_EAS_NOT_SUPPORTED:
        Win32ErrorCodeDescription :=
            'The mounted file system does not support extended attributes.';
    Win32ErrorCodes.ERROR_NOT_OWNER:
        Win32ErrorCodeDescription := 'Attempt to release mutex not owned by caller.';
    Win32ErrorCodes.ERROR_TOO_MANY_POSTS:
        Win32ErrorCodeDescription := 'Too many posts were made to a semaphore.';
    Win32ErrorCodes.ERROR_PARTIAL_COPY:
        Win32ErrorCodeDescription :=
            'Only part of a ReadProcessMemory or WriteProcessMemory request was completed.';
    Win32ErrorCodes.ERROR_OPLOCK_NOT_GRANTED:
        Win32ErrorCodeDescription := 'The oplock request is denied.';
    Win32ErrorCodes.ERROR_INVALID_OPLOCK_PROTOCOL:
        Win32ErrorCodeDescription :=
            'An invalid oplock acknowledgment was received by the system.';
    Win32ErrorCodes.ERROR_DISK_TOO_FRAGMENTED:
        Win32ErrorCodeDescription := 'The volume is too fragmented to complete this operation.';
    Win32ErrorCodes.ERROR_DELETE_PENDING:
        Win32ErrorCodeDescription :=
            'The file cannot be opened because it is in the process of being deleted.';
    Win32ErrorCodes.ERROR_MR_MID_NOT_FOUND:
        Win32ErrorCodeDescription :=
            'The system cannot find message text for message number 0x%1 in the message file for %2.';
    Win32ErrorCodes.ERROR_INVALID_ADDRESS:
        Win32ErrorCodeDescription := 'Attempt to access invalid address.';
    Win32ErrorCodes.ERROR_ARITHMETIC_OVERFLOW:
        Win32ErrorCodeDescription := 'Arithmetic result exceeded 32 bits.';
    Win32ErrorCodes.ERROR_PIPE_CONNECTED:
        Win32ErrorCodeDescription := 'There is a process on other end of the pipe.';
    Win32ErrorCodes.ERROR_PIPE_LISTENING:
        Win32ErrorCodeDescription := 'Waiting for a process to open the other end of the pipe.';
    Win32ErrorCodes.ERROR_EA_ACCESS_DENIED:
        Win32ErrorCodeDescription := 'Access to the extended attribute was denied.';
    Win32ErrorCodes.ERROR_OPERATION_ABORTED:
        Win32ErrorCodeDescription := 'The I/O operation has been aborted because of either a thread exit or an application request.';
    Win32ErrorCodes.ERROR_IO_INCOMPLETE:
        Win32ErrorCodeDescription := 'Overlapped I/O event is not in a signaled state.';
    Win32ErrorCodes.ERROR_IO_PENDING:
        Win32ErrorCodeDescription := 'Overlapped I/O operation is in progress.';
    Win32ErrorCodes.ERROR_NOACCESS:
        Win32ErrorCodeDescription := 'Invalid access to memory location.';
    Win32ErrorCodes.ERROR_SWAPERROR:
        Win32ErrorCodeDescription := 'Error performing inpage operation.';
    Win32ErrorCodes.ERROR_STACK_OVERFLOW:
        Win32ErrorCodeDescription := 'Recursion too deep; the stack overflowed.';
    Win32ErrorCodes.ERROR_INVALID_MESSAGE:
        Win32ErrorCodeDescription := 'The window cannot act on the sent message.';
    Win32ErrorCodes.ERROR_CAN_NOT_COMPLETE:
        Win32ErrorCodeDescription := 'Cannot complete this function.';
    Win32ErrorCodes.ERROR_INVALID_FLAGS:
        Win32ErrorCodeDescription := 'Invalid flags.';
    Win32ErrorCodes.ERROR_UNRECOGNIZED_VOLUME:
        Win32ErrorCodeDescription := 'The volume does not contain a recognized file system. Please make sure that all required file system drivers are loaded and that the volume is not corrupted.';
    Win32ErrorCodes.ERROR_FILE_INVALID:
        Win32ErrorCodeDescription := 'The volume for a file has been externally altered so that the opened file is no longer valid.';
    Win32ErrorCodes.ERROR_FULLSCREEN_MODE:
        Win32ErrorCodeDescription :=
            'The requested operation cannot be performed in full-screen mode.';
    Win32ErrorCodes.ERROR_NO_TOKEN:
        Win32ErrorCodeDescription :=
            'An attempt was made to reference a token that does not exist.';
    Win32ErrorCodes.ERROR_BADDB:
        Win32ErrorCodeDescription := 'The configuration registry database is corrupt.';
    Win32ErrorCodes.ERROR_BADKEY:
        Win32ErrorCodeDescription := 'The configuration registry key is invalid.';
    Win32ErrorCodes.ERROR_CANTOPEN:
        Win32ErrorCodeDescription := 'The configuration registry key could not be opened.';
    Win32ErrorCodes.ERROR_CANTREAD:
        Win32ErrorCodeDescription := 'The configuration registry key could not be read.';
    Win32ErrorCodes.ERROR_CANTWRITE:
        Win32ErrorCodeDescription := 'The configuration registry key could not be written.';
    Win32ErrorCodes.ERROR_REGISTRY_RECOVERED:
        Win32ErrorCodeDescription := 'One of the files in the registry database had to be recovered by use of a log or alternate copy. The recovery was successful.';
    Win32ErrorCodes.ERROR_REGISTRY_CORRUPT:
        Win32ErrorCodeDescription := 'The registry is corrupted. The structure of one of the files containing registry data is corrupted, or the systems memory image of the file is corrupted, or the file could not be recovered because the alternate copy or log was absent or corrupted.';
    Win32ErrorCodes.ERROR_REGISTRY_IO_FAILED:
        Win32ErrorCodeDescription := 'An I/O operation initiated by the registry failed unrecoverably. The registry could not read in, or write out, or flush, one of the files that contain the systems image of the registry.';
    Win32ErrorCodes.ERROR_NOT_REGISTRY_FILE:
        Win32ErrorCodeDescription := 'The system has attempted to load or restore a file into the registry, but the specified file is not in a registry file format.';
    Win32ErrorCodes.ERROR_KEY_DELETED:
        Win32ErrorCodeDescription :=
            'Illegal operation attempted on a registry key that has been marked for deletion.';
    Win32ErrorCodes.ERROR_NO_LOG_SPACE:
        Win32ErrorCodeDescription :=
            'System could not allocate the required space in a registry log.';
    Win32ErrorCodes.ERROR_KEY_HAS_CHILDREN:
        Win32ErrorCodeDescription :=
            'Cannot create a symbolic link in a registry key that already has subkeys or values.';
    Win32ErrorCodes.ERROR_CHILD_MUST_BE_VOLATILE:
        Win32ErrorCodeDescription := 'Cannot create a stable subkey under a volatile parent key.';
    Win32ErrorCodes.ERROR_NOTIFY_ENUM_DIR:
        Win32ErrorCodeDescription := 'A notify change request is being completed and the information is not being returned in the callers buffer. The caller now needs to enumerate the files to find the changes.';
    Win32ErrorCodes.ERROR_DEPENDENT_SERVICES_RUNNING:
        Win32ErrorCodeDescription :=
            'A stop control has been sent to a service that other running services are dependent on.';
    Win32ErrorCodes.ERROR_INVALID_SERVICE_CONTROL:
        Win32ErrorCodeDescription := 'The requested control is not valid for this service.';
    Win32ErrorCodes.ERROR_SERVICE_REQUEST_TIMEOUT:
        Win32ErrorCodeDescription :=
            'The service did not respond to the start or control request in a timely fashion.';
    Win32ErrorCodes.ERROR_SERVICE_NO_THREAD:
        Win32ErrorCodeDescription := 'A thread could not be created for the service.';
    Win32ErrorCodes.ERROR_SERVICE_DATABASE_LOCKED:
        Win32ErrorCodeDescription := 'The service database is locked.';
    Win32ErrorCodes.ERROR_SERVICE_ALREADY_RUNNING:
        Win32ErrorCodeDescription := 'An instance of the service is already running.';
    Win32ErrorCodes.ERROR_INVALID_SERVICE_ACCOUNT:
        Win32ErrorCodeDescription := 'The account name is invalid or does not exist, or the password is invalid for the account name specified.';
    Win32ErrorCodes.ERROR_SERVICE_DISABLED:
        Win32ErrorCodeDescription := 'The service cannot be started, either because it is disabled or because it has no enabled devices associated with it.';
    Win32ErrorCodes.ERROR_CIRCULAR_DEPENDENCY:
        Win32ErrorCodeDescription := 'Circular service dependency was specified.';
    Win32ErrorCodes.ERROR_SERVICE_DOES_NOT_EXIST:
        Win32ErrorCodeDescription :=
            'The specified service does not exist as an installed service.';
    Win32ErrorCodes.ERROR_SERVICE_CANNOT_ACCEPT_CTRL:
        Win32ErrorCodeDescription := 'The service cannot accept control messages at this time.';
    Win32ErrorCodes.ERROR_SERVICE_NOT_ACTIVE:
        Win32ErrorCodeDescription := 'The service has not been started.';
    Win32ErrorCodes.ERROR_FAILED_SERVICE_CONTROLLER_CONNECT:
        Win32ErrorCodeDescription :=
            'The service process could not connect to the service controller.';
    Win32ErrorCodes.ERROR_EXCEPTION_IN_SERVICE:
        Win32ErrorCodeDescription :=
            'An exception occurred in the service when handling the control request.';
    Win32ErrorCodes.ERROR_DATABASE_DOES_NOT_EXIST:
        Win32ErrorCodeDescription := 'The database specified does not exist.';
    Win32ErrorCodes.ERROR_SERVICE_SPECIFIC_ERROR:
        Win32ErrorCodeDescription := 'The service has returned a service-specific error code.';
    Win32ErrorCodes.ERROR_PROCESS_ABORTED:
        Win32ErrorCodeDescription := 'The process terminated unexpectedly.';
    Win32ErrorCodes.ERROR_SERVICE_DEPENDENCY_FAIL:
        Win32ErrorCodeDescription := 'The dependency service or group failed to start.';
    Win32ErrorCodes.ERROR_SERVICE_LOGON_FAILED:
        Win32ErrorCodeDescription := 'The service did not start due to a logon failure.';
    Win32ErrorCodes.ERROR_SERVICE_START_HANG:
        Win32ErrorCodeDescription := 'After starting, the service hung in a start-pending state.';
    Win32ErrorCodes.ERROR_INVALID_SERVICE_LOCK:
        Win32ErrorCodeDescription := 'The specified service database lock is invalid.';
    Win32ErrorCodes.ERROR_SERVICE_MARKED_FOR_DELETE:
        Win32ErrorCodeDescription := 'The specified service has been marked for deletion.';
    Win32ErrorCodes.ERROR_SERVICE_EXISTS:
        Win32ErrorCodeDescription := 'The specified service already exists.';
    Win32ErrorCodes.ERROR_ALREADY_RUNNING_LKG:
        Win32ErrorCodeDescription :=
            'The system is currently running with the last-known-good configuration.';
    Win32ErrorCodes.ERROR_SERVICE_DEPENDENCY_DELETED:
        Win32ErrorCodeDescription :=
            'The dependency service does not exist or has been marked for deletion.';
    Win32ErrorCodes.ERROR_BOOT_ALREADY_ACCEPTED:
        Win32ErrorCodeDescription :=
            'The current boot has already been accepted for use as the last-known-good control set.';
    Win32ErrorCodes.ERROR_SERVICE_NEVER_STARTED:
        Win32ErrorCodeDescription :=
            'No attempts to start the service have been made since the last boot.';
    Win32ErrorCodes.ERROR_DUPLICATE_SERVICE_NAME:
        Win32ErrorCodeDescription :=
            'The name is already in use as either a service name or a service display name.';
    Win32ErrorCodes.ERROR_DIFFERENT_SERVICE_ACCOUNT:
        Win32ErrorCodeDescription := 'The account specified for this service is different from the account specified for other services running in the same process.';
    Win32ErrorCodes.ERROR_CANNOT_DETECT_DRIVER_FAILURE:
        Win32ErrorCodeDescription :=
            'Failure actions can only be set for Win32 services, not for drivers.';
    Win32ErrorCodes.ERROR_CANNOT_DETECT_PROCESS_ABORT:
        Win32ErrorCodeDescription := 'This service runs in the same process as the service control manager. Therefore, the service control manager cannot take action if this services process terminates unexpectedly.';
    Win32ErrorCodes.ERROR_NO_RECOVERY_PROGRAM:
        Win32ErrorCodeDescription := 'No recovery program has been configured for this service.';
    Win32ErrorCodes.ERROR_SERVICE_NOT_IN_EXE:
        Win32ErrorCodeDescription := 'The executable program that this service is configured to run in does not implement the service.';
    Win32ErrorCodes.ERROR_NOT_SAFEBOOT_SERVICE:
        Win32ErrorCodeDescription := 'This service cannot be started in Safe Mode.';
    Win32ErrorCodes.ERROR_END_OF_MEDIA:
        Win32ErrorCodeDescription := 'The physical end of the tape has been reached.';
    Win32ErrorCodes.ERROR_FILEMARK_DETECTED:
        Win32ErrorCodeDescription := 'A tape access reached a filemark.';
    Win32ErrorCodes.ERROR_BEGINNING_OF_MEDIA:
        Win32ErrorCodeDescription := 'The beginning of the tape or a partition was encountered.';
    Win32ErrorCodes.ERROR_SETMARK_DETECTED:
        Win32ErrorCodeDescription := 'A tape access reached the end of a set of files.';
    Win32ErrorCodes.ERROR_NO_DATA_DETECTED:
        Win32ErrorCodeDescription := 'No more data is on the tape.';
    Win32ErrorCodes.ERROR_PARTITION_FAILURE:
        Win32ErrorCodeDescription := 'Tape could not be partitioned.';
    Win32ErrorCodes.ERROR_INVALID_BLOCK_LENGTH:
        Win32ErrorCodeDescription := 'When accessing a new tape of a multivolume partition, the current block size is incorrect.';
    Win32ErrorCodes.ERROR_DEVICE_NOT_PARTITIONED:
        Win32ErrorCodeDescription :=
            'Tape partition information could not be found when loading a tape.';
    Win32ErrorCodes.ERROR_UNABLE_TO_LOCK_MEDIA:
        Win32ErrorCodeDescription := 'Unable to lock the media eject mechanism.';
    Win32ErrorCodes.ERROR_UNABLE_TO_UNLOAD_MEDIA:
        Win32ErrorCodeDescription := 'Unable to unload the media.';
    Win32ErrorCodes.ERROR_MEDIA_CHANGED:
        Win32ErrorCodeDescription := 'The media in the drive may have changed.';
    Win32ErrorCodes.ERROR_BUS_RESET:
        Win32ErrorCodeDescription := 'The I/O bus was reset.';
    Win32ErrorCodes.ERROR_NO_MEDIA_IN_DRIVE:
        Win32ErrorCodeDescription := 'No media in drive.';
    Win32ErrorCodes.ERROR_NO_UNICODE_TRANSLATION:
        Win32ErrorCodeDescription :=
            'No mapping for the Unicode character exists in the target multi-byte code page.';
    Win32ErrorCodes.ERROR_DLL_INIT_FAILED:
        Win32ErrorCodeDescription := 'A dynamic link library (DLL) initialization routine failed.';
    Win32ErrorCodes.ERROR_SHUTDOWN_IN_PROGRESS:
        Win32ErrorCodeDescription := 'A system shutdown is in progress.';
    Win32ErrorCodes.ERROR_NO_SHUTDOWN_IN_PROGRESS:
        Win32ErrorCodeDescription :=
            'Unable to abort the system shutdown because no shutdown was in progress.';
    Win32ErrorCodes.ERROR_IO_DEVICE:
        Win32ErrorCodeDescription :=
            'The request could not be performed because of an I/O device error.';
    Win32ErrorCodes.ERROR_SERIAL_NO_DEVICE:
        Win32ErrorCodeDescription :=
            'No serial device was successfully initialized. The serial driver will unload.';
    Win32ErrorCodes.ERROR_IRQ_BUSY:
        Win32ErrorCodeDescription := 'Unable to open a device that was sharing an interrupt request (IRQ) with other devices. At least one other device that uses that IRQ was already opened.';
    Win32ErrorCodes.ERROR_MORE_WRITES:
        Win32ErrorCodeDescription := 'A serial I/O operation was completed by another write to the serial port. (The IOCTL_SERIAL_XOFF_COUNTER reached zero.)';
    Win32ErrorCodes.ERROR_COUNTER_TIMEOUT:
        Win32ErrorCodeDescription := 'A serial I/O operation completed because the timeout period expired. (The IOCTL_SERIAL_XOFF_COUNTER did not reach zero.)';
    Win32ErrorCodes.ERROR_FLOPPY_ID_MARK_NOT_FOUND:
        Win32ErrorCodeDescription := 'No ID address mark was found on the floppy disk.';
    Win32ErrorCodes.ERROR_FLOPPY_WRONG_CYLINDER:
        Win32ErrorCodeDescription := 'Mismatch between the floppy disk sector ID field and the floppy disk controller track address.';
    Win32ErrorCodes.ERROR_FLOPPY_UNKNOWN_ERROR:
        Win32ErrorCodeDescription := 'The floppy disk controller reported an error that is not recognized by the floppy disk driver.';
    Win32ErrorCodes.ERROR_FLOPPY_BAD_REGISTERS:
        Win32ErrorCodeDescription :=
            'The floppy disk controller returned inconsistent results in its registers.';
    Win32ErrorCodes.ERROR_DISK_RECALIBRATE_FAILED:
        Win32ErrorCodeDescription :=
            'While accessing the hard disk, a recalibrate operation failed, even after retries.';
    Win32ErrorCodes.ERROR_DISK_OPERATION_FAILED:
        Win32ErrorCodeDescription :=
            'While accessing the hard disk, a disk operation failed even after retries.';
    Win32ErrorCodes.ERROR_DISK_RESET_FAILED:
        Win32ErrorCodeDescription :=
            'While accessing the hard disk, a disk controller reset was needed, but even that failed.';
    Win32ErrorCodes.ERROR_EOM_OVERFLOW:
        Win32ErrorCodeDescription := 'Physical end of tape encountered.';
    Win32ErrorCodes.ERROR_NOT_ENOUGH_SERVER_MEMORY:
        Win32ErrorCodeDescription :=
            'Not enough server storage is available to process this command.';
    Win32ErrorCodes.ERROR_POSSIBLE_DEADLOCK:
        Win32ErrorCodeDescription := 'A potential deadlock condition has been detected.';
    Win32ErrorCodes.ERROR_MAPPED_ALIGNMENT:
        Win32ErrorCodeDescription :=
            'The base address or the file offset specified does not have the proper alignment.';
    Win32ErrorCodes.ERROR_SET_POWER_STATE_VETOED:
        Win32ErrorCodeDescription :=
            'An attempt to change the system power state was vetoed by another application or driver.';
    Win32ErrorCodes.ERROR_SET_POWER_STATE_FAILED:
        Win32ErrorCodeDescription :=
            'The system BIOS failed an attempt to change the system power state.';
    Win32ErrorCodes.ERROR_TOO_MANY_LINKS:
        Win32ErrorCodeDescription :=
            'An attempt was made to create more links on a file than the file system supports.';
    Win32ErrorCodes.ERROR_OLD_WIN_VERSION:
        Win32ErrorCodeDescription := 'The specified program requires a newer version of Windows.';
    Win32ErrorCodes.ERROR_APP_WRONG_OS:
        Win32ErrorCodeDescription := 'The specified program is not a Windows or MS-DOS program.';
    Win32ErrorCodes.ERROR_SINGLE_INSTANCE_APP:
        Win32ErrorCodeDescription :=
            'Cannot start more than one instance of the specified program.';
    Win32ErrorCodes.ERROR_RMODE_APP:
        Win32ErrorCodeDescription :=
            'The specified program was written for an earlier version of Windows.';
    Win32ErrorCodes.ERROR_INVALID_DLL:
        Win32ErrorCodeDescription :=
            'One of the library files needed to run this application is damaged.';
    Win32ErrorCodes.ERROR_NO_ASSOCIATION:
        Win32ErrorCodeDescription :=
            'No application is associated with the specified file for this operation.';
    Win32ErrorCodes.ERROR_DDE_FAIL:
        Win32ErrorCodeDescription :=
            'An error occurred in sending the command to the application.';
    Win32ErrorCodes.ERROR_DLL_NOT_FOUND:
        Win32ErrorCodeDescription :=
            'One of the library files needed to run this application cannot be found.';
    Win32ErrorCodes.ERROR_NO_MORE_USER_HANDLES:
        Win32ErrorCodeDescription := 'The current process has used all of its system allowance of handles for Window Manager objects.';
    Win32ErrorCodes.ERROR_MESSAGE_SYNC_ONLY:
        Win32ErrorCodeDescription := 'The message can be used only with synchronous operations.';
    Win32ErrorCodes.ERROR_SOURCE_ELEMENT_EMPTY:
        Win32ErrorCodeDescription := 'The indicated source element has no media.';
    Win32ErrorCodes.ERROR_DESTINATION_ELEMENT_FULL:
        Win32ErrorCodeDescription := 'The indicated destination element already contains media.';
    Win32ErrorCodes.ERROR_ILLEGAL_ELEMENT_ADDRESS:
        Win32ErrorCodeDescription := 'The indicated element does not exist.';
    Win32ErrorCodes.ERROR_MAGAZINE_NOT_PRESENT:
        Win32ErrorCodeDescription :=
            'The indicated element is part of a magazine that is not present.';
    Win32ErrorCodes.ERROR_DEVICE_REINITIALIZATION_NEEDED:
        Win32ErrorCodeDescription :=
            'The indicated device requires reinitialization due to hardware errors.';
    Win32ErrorCodes.ERROR_DEVICE_REQUIRES_CLEANING:
        Win32ErrorCodeDescription := 'The device has indicated that cleaning is required before further operations are attempted.';
    Win32ErrorCodes.ERROR_DEVICE_DOOR_OPEN:
        Win32ErrorCodeDescription := 'The device has indicated that its door is open.';
    Win32ErrorCodes.ERROR_DEVICE_NOT_CONNECTED:
        Win32ErrorCodeDescription := 'The device is not connected.';
    Win32ErrorCodes.ERROR_NOT_FOUND:
        Win32ErrorCodeDescription := 'Element not found.';
    Win32ErrorCodes.ERROR_NO_MATCH:
        Win32ErrorCodeDescription := 'There was no match for the specified key in the index.';
    Win32ErrorCodes.ERROR_SET_NOT_FOUND:
        Win32ErrorCodeDescription := 'The property set specified does not exist on the object.';
    Win32ErrorCodes.ERROR_POINT_NOT_FOUND:
        Win32ErrorCodeDescription :=
            'The point passed to GetMouseMovePointsEx is not in the buffer.';
    Win32ErrorCodes.ERROR_NO_TRACKING_SERVICE:
        Win32ErrorCodeDescription := 'The tracking (workstation) service is not running.';
    Win32ErrorCodes.ERROR_NO_VOLUME_ID:
        Win32ErrorCodeDescription := 'The Volume ID could not be found.';
    Win32ErrorCodes.ERROR_UNABLE_TO_REMOVE_REPLACED:
        Win32ErrorCodeDescription := 'Unable to remove the file to be replaced.';
    Win32ErrorCodes.ERROR_UNABLE_TO_MOVE_REPLACEMENT:
        Win32ErrorCodeDescription := 'Unable to move the replacement file to the file to be replaced. The file to be replaced has retained its original name.';
    Win32ErrorCodes.ERROR_UNABLE_TO_MOVE_REPLACEMENT_2:
        Win32ErrorCodeDescription := 'Unable to move the replacement file to the file to be replaced. The file to be replaced has been renamed using the backup name.';
    Win32ErrorCodes.ERROR_JOURNAL_DELETE_IN_PROGRESS:
        Win32ErrorCodeDescription := 'The volume change journal is being deleted.';
    Win32ErrorCodes.ERROR_JOURNAL_NOT_ACTIVE:
        Win32ErrorCodeDescription := 'The volume change journal is not active.';
    Win32ErrorCodes.ERROR_POTENTIAL_FILE_FOUND:
        Win32ErrorCodeDescription := 'A file was found, but it may not be the correct file.';
    Win32ErrorCodes.ERROR_JOURNAL_ENTRY_DELETED:
        Win32ErrorCodeDescription := 'The journal entry has been deleted from the journal.';
    Win32ErrorCodes.ERROR_BAD_DEVICE:
        Win32ErrorCodeDescription := 'The specified device name is invalid.';
    Win32ErrorCodes.ERROR_CONNECTION_UNAVAIL:
        Win32ErrorCodeDescription :=
            'The device is not currently connected but it is a remembered connection.';
    Win32ErrorCodes.ERROR_DEVICE_ALREADY_REMEMBERED:
        Win32ErrorCodeDescription :=
            'The local device name has a remembered connection to another network resource.';
    Win32ErrorCodes.ERROR_NO_NET_OR_BAD_PATH:
        Win32ErrorCodeDescription := 'No network provider accepted the given network path.';
    Win32ErrorCodes.ERROR_BAD_PROVIDER:
        Win32ErrorCodeDescription := 'The specified network provider name is invalid.';
    Win32ErrorCodes.ERROR_CANNOT_OPEN_PROFILE:
        Win32ErrorCodeDescription := 'Unable to open the network connection profile.';
    Win32ErrorCodes.ERROR_BAD_PROFILE:
        Win32ErrorCodeDescription := 'The network connection profile is corrupted.';
    Win32ErrorCodes.ERROR_NOT_CONTAINER:
        Win32ErrorCodeDescription := 'Cannot enumerate a noncontainer.';
    Win32ErrorCodes.ERROR_EXTENDED_ERROR:
        Win32ErrorCodeDescription := 'An extended error has occurred.';
    Win32ErrorCodes.ERROR_INVALID_GROUPNAME:
        Win32ErrorCodeDescription := 'The format of the specified group name is invalid.';
    Win32ErrorCodes.ERROR_INVALID_COMPUTERNAME:
        Win32ErrorCodeDescription := 'The format of the specified computer name is invalid.';
    Win32ErrorCodes.ERROR_INVALID_EVENTNAME:
        Win32ErrorCodeDescription := 'The format of the specified event name is invalid.';
    Win32ErrorCodes.ERROR_INVALID_DOMAINNAME:
        Win32ErrorCodeDescription := 'The format of the specified domain name is invalid.';
    Win32ErrorCodes.ERROR_INVALID_SERVICENAME:
        Win32ErrorCodeDescription := 'The format of the specified service name is invalid.';
    Win32ErrorCodes.ERROR_INVALID_NETNAME:
        Win32ErrorCodeDescription := 'The format of the specified network name is invalid.';
    Win32ErrorCodes.ERROR_INVALID_SHARENAME:
        Win32ErrorCodeDescription := 'The format of the specified share name is invalid.';
    Win32ErrorCodes.ERROR_INVALID_PASSWORDNAME:
        Win32ErrorCodeDescription := 'The format of the specified password is invalid.';
    Win32ErrorCodes.ERROR_INVALID_MESSAGENAME:
        Win32ErrorCodeDescription := 'The format of the specified message name is invalid.';
    Win32ErrorCodes.ERROR_INVALID_MESSAGEDEST:
        Win32ErrorCodeDescription := 'The format of the specified message destination is invalid.';
    Win32ErrorCodes.ERROR_SESSION_CREDENTIAL_CONFLICT:
        Win32ErrorCodeDescription :=
            'The credentials supplied conflict with an existing set of credentials.';
    Win32ErrorCodes.ERROR_REMOTE_SESSION_LIMIT_EXCEEDED:
        Win32ErrorCodeDescription := 'An attempt was made to establish a session to a network server, but there are already too many sessions established to that server.';
    Win32ErrorCodes.ERROR_DUP_DOMAINNAME:
        Win32ErrorCodeDescription :=
            'The workgroup or domain name is already in use by another computer on the network.';
    Win32ErrorCodes.ERROR_NO_NETWORK:
        Win32ErrorCodeDescription := 'The network is not present or not started.';
    Win32ErrorCodes.ERROR_CANCELLED:
        Win32ErrorCodeDescription := 'The operation was canceled by the user.';
    Win32ErrorCodes.ERROR_USER_MAPPED_FILE:
        Win32ErrorCodeDescription :=
            'The requested operation cannot be performed on a file with a user-mapped section open.';
    Win32ErrorCodes.ERROR_CONNECTION_REFUSED:
        Win32ErrorCodeDescription := 'The remote system refused the network connection.';
    Win32ErrorCodes.ERROR_GRACEFUL_DISCONNECT:
        Win32ErrorCodeDescription := 'The network connection was gracefully closed.';
    Win32ErrorCodes.ERROR_ADDRESS_ALREADY_ASSOCIATED:
        Win32ErrorCodeDescription :=
            'The network transport endpoint already has an address associated with it.';
    Win32ErrorCodes.ERROR_ADDRESS_NOT_ASSOCIATED:
        Win32ErrorCodeDescription :=
            'An address has not yet been associated with the network endpoint.';
    Win32ErrorCodes.ERROR_CONNECTION_INVALID:
        Win32ErrorCodeDescription :=
            'An operation was attempted on a nonexistent network connection.';
    Win32ErrorCodes.ERROR_CONNECTION_ACTIVE:
        Win32ErrorCodeDescription :=
            'An invalid operation was attempted on an active network connection.';
    Win32ErrorCodes.ERROR_NETWORK_UNREACHABLE:
        Win32ErrorCodeDescription := 'The network location cannot be reached. For information about network troubleshooting, see Windows Help.';
    Win32ErrorCodes.ERROR_HOST_UNREACHABLE:
        Win32ErrorCodeDescription := 'The network location cannot be reached. For information about network troubleshooting, see Windows Help.';
    Win32ErrorCodes.ERROR_PROTOCOL_UNREACHABLE:
        Win32ErrorCodeDescription := 'The network location cannot be reached. For information about network troubleshooting, see Windows Help.';
    Win32ErrorCodes.ERROR_PORT_UNREACHABLE:
        Win32ErrorCodeDescription :=
            'No service is operating at the destination network endpoint on the remote system.';
    Win32ErrorCodes.ERROR_REQUEST_ABORTED:
        Win32ErrorCodeDescription := 'The request was aborted.';
    Win32ErrorCodes.ERROR_CONNECTION_ABORTED:
        Win32ErrorCodeDescription := 'The network connection was aborted by the local system.';
    Win32ErrorCodes.ERROR_RETRY:
        Win32ErrorCodeDescription :=
            'The operation could not be completed. A retry should be performed.';
    Win32ErrorCodes.ERROR_CONNECTION_COUNT_LIMIT:
        Win32ErrorCodeDescription := 'A connection to the server could not be made because the limit on the number of concurrent connections for this account has been reached.';
    Win32ErrorCodes.ERROR_LOGIN_TIME_RESTRICTION:
        Win32ErrorCodeDescription :=
            'Attempting to log in during an unauthorized time of day for this account.';
    Win32ErrorCodes.ERROR_LOGIN_WKSTA_RESTRICTION:
        Win32ErrorCodeDescription := 'The account is not authorized to log in from this station.';
    Win32ErrorCodes.ERROR_INCORRECT_ADDRESS:
        Win32ErrorCodeDescription :=
            'The network address could not be used for the operation requested.';
    Win32ErrorCodes.ERROR_ALREADY_REGISTERED:
        Win32ErrorCodeDescription := 'The service is already registered.';
    Win32ErrorCodes.ERROR_SERVICE_NOT_FOUND:
        Win32ErrorCodeDescription := 'The specified service does not exist.';
    Win32ErrorCodes.ERROR_NOT_AUTHENTICATED:
        Win32ErrorCodeDescription := 'The operation being requested was not performed because the user has not been authenticated.';
    Win32ErrorCodes.ERROR_NOT_LOGGED_ON:
        Win32ErrorCodeDescription := 'The operation being requested was not performed because the user has not logged on to the network. The specified service does not exist.';
    Win32ErrorCodes.ERROR_CONTINUE:
        Win32ErrorCodeDescription := 'Continue with work in progress.';
    Win32ErrorCodes.ERROR_ALREADY_INITIALIZED:
        Win32ErrorCodeDescription := 'An attempt was made to perform an initialization operation when initialization has already been completed.';
    Win32ErrorCodes.ERROR_NO_MORE_DEVICES:
        Win32ErrorCodeDescription := 'No more local devices.';
    Win32ErrorCodes.ERROR_NO_SUCH_SITE:
        Win32ErrorCodeDescription := 'The specified site does not exist.';
    Win32ErrorCodes.ERROR_DOMAIN_CONTROLLER_EXISTS:
        Win32ErrorCodeDescription := 'A domain controller with the specified name already exists.';
    Win32ErrorCodes.ERROR_ONLY_IF_CONNECTED:
        Win32ErrorCodeDescription :=
            'This operation is supported only when you are connected to the server.';
    Win32ErrorCodes.ERROR_OVERRIDE_NOCHANGES:
        Win32ErrorCodeDescription :=
            'The group policy framework should call the extension even if there are no changes.';
    Win32ErrorCodes.ERROR_BAD_USER_PROFILE:
        Win32ErrorCodeDescription := 'The specified user does not have a valid profile.';
    Win32ErrorCodes.ERROR_NOT_SUPPORTED_ON_SBS:
        Win32ErrorCodeDescription :=
            'This operation is not supported on a Microsoft Small Business Server.';
    Win32ErrorCodes.ERROR_SERVER_SHUTDOWN_IN_PROGRESS:
        Win32ErrorCodeDescription := 'The server machine is shutting down.';
    Win32ErrorCodes.ERROR_HOST_DOWN:
        Win32ErrorCodeDescription := 'The remote system is not available. For information about network troubleshooting, see Windows Help.';
    Win32ErrorCodes.ERROR_NON_ACCOUNT_SID:
        Win32ErrorCodeDescription :=
            'The security identifier provided is not from an account domain.';
    Win32ErrorCodes.ERROR_NON_DOMAIN_SID:
        Win32ErrorCodeDescription :=
            'The security identifier provided does not have a domain component.';
    Win32ErrorCodes.ERROR_APPHELP_BLOCK:
        Win32ErrorCodeDescription :=
            'AppHelp dialog canceled thus preventing the application from starting.';
    Win32ErrorCodes.ERROR_ACCESS_DISABLED_BY_POLICY:
        Win32ErrorCodeDescription :=
            'Access to the requested resource has been disabled by your administrator.';
    Win32ErrorCodes.ERROR_REG_NAT_CONSUMPTION:
        Win32ErrorCodeDescription := 'A program attempt to use an invalid register value. Normally caused by an uninitialized register. This error is Itanium specific.';
    Win32ErrorCodes.ERROR_CSCSHARE_OFFLINE:
        Win32ErrorCodeDescription := 'The share is currently offline or does not exist.';
    Win32ErrorCodes.ERROR_NOT_ALL_ASSIGNED:
        Win32ErrorCodeDescription := 'Not all privileges referenced are assigned to the caller.';
    Win32ErrorCodes.ERROR_SOME_NOT_MAPPED:
        Win32ErrorCodeDescription :=
            'Some mapping between account names and security IDs was not done.';
    Win32ErrorCodes.ERROR_NO_QUOTAS_FOR_ACCOUNT:
        Win32ErrorCodeDescription :=
            'No system quota limits are specifically set for this account.';
    Win32ErrorCodes.ERROR_LOCAL_USER_SESSION_KEY:
        Win32ErrorCodeDescription :=
            'No encryption key is available. A well-known encryption key was returned.';
    Win32ErrorCodes.ERROR_NULL_LM_PASSWORD:
